    def main_calculate_step_left(p11, p12, p21, p22, p3, p13, p23, noncappingsidewallthick, cappingsidewallthick, tcp_pose_top):
        struct1 = analyze_touchpoints_only(p11, p12, p21, p22, p3)
        list1 = analyze_vertical_touchpoints(p11, p12, p13, p21, p22, p23, p3)
        #struct2 = calculate_DOtA_points_right(struct1, list1, chamferover)
        #validity = check_validity_right(struct1, struct2)
        struct2 = calculate_DAaU_step_left(struct1, list1, cappingsidewallthick, noncappingsidewallthick, tcp_pose_top)
        validity = check_validity_only(struct2)
        return struct2
    end

    # analyze_touchpoints_only()
    # it takes 5 arguments as points
    # it returns a struct containing: (pointintersect, heading1, heading2, heading3, l1delxunit, l1delyunit, l2delxunit, l2delyunit)
    #   FIND HEADINGS
    #for each heading, find the angle of the line with respect to the pos x axis. then add/subtract 90 degrees because you want to be perpendicular to that
    # so, heading1 finds the angle (from the +x axis) to the position pointing perpendicularly into the box.
    # we need to be +90 degrees of all 3 headings. (but we can ignore heading 2)
    def step_right_demo(struct1):
        pointintersect = struct1[0]
        x = pointintersect[0]
        y = pointintersect[1]
        z = pointintersect[2]
        heading1 = struct1[1]
        heading1adj1 = heading1 + pi/2 #(90 deg) (parrallel to edge not perpendicular into
        heading1adj2 = heading1adj1 - pi/2 #(90 deg) (from y+ not x+)
        # heading1 == heading1adj2. ok
        m1 = get_rotation_matrix_from_description("z", 1, heading1)
        # at this point we would multiply matrices, but there is only one matrix
        rxryrz = convert_matrix_to_axang(m1)
        point_demo = p[x, y, z, rxryrz[0], rxryrz[1], rxryrz[2]]
        popup(point_demo)
        movej(point_demo, a=1.4, v=0.1)
        popup(point_demo)
        ret = struct(point_demo = point_demo)
        return ret
    end

    # for a left seam step corner, calculate the toolpath points for a L (under) then Up and Around weld. for left obstacle step.
    def calculate_LtUA_step_left(struct1, listleans, rightwallthick, leftwallthick, tcp_pose_top):
        # get the stuff from the struct
        pointintersect = struct1[0]
        heading1 = struct1[1]
        heading2 = struct1[2]
        heading3 = struct1[3]
        l1delxunit = struct1[4]
        l1delyunit = struct1[5]
        l2delxunit = struct1[6]
        l2delyunit = struct1[7]

        # FIND THE POINTS ON THE LINES OF THE FIRST TURN PATH
        # find locations 8 inches away from  intersect point
        # CONST
        welddistance1 = 3 # first path first leg
        welddistance2 = 3 # first path second leg
        welddistance3 = 8 # vertical weld distance

        # inches
        wd1 = welddistance1 * 25.4 / 1000
        wd2 = welddistance2 * 25.4 / 1000
        wd3 = tcp_pose_top[2] - pointintersect[2] # the z distance from the corner to the top of the weld
        leftwallthickmm = leftwallthick * 25.4 / 1000 # in this step corner right, this is distance from left edge
        rightwallthickmm =  rightwallthick * 25.4 / 1000 # in this step corner right, this is distance from right edge


        # weld distance is the distance that it will weld. this will make it start at the z height that the user specified
        #wd1 = tcp_pose_top[2] - pointintersect[2] - zup # this will need to change for step corner right

        # point bottom (point of intersection of the two chamfers on the bottom)
        xbottom = pointintersect[0] + l1delxunit * leftwallthickmm + l2delxunit * rightwallthickmm
        ybottom = pointintersect[1] + l1delyunit * leftwallthickmm + l2delyunit * rightwallthickmm
        z = pointintersect[2]

        # point 1
        x = xbottom + l1delxunit * wd1
        y = ybottom + l1delyunit * wd1

        # get rxryrz for facing along towards the intersection. heading1 +90 deg - 90 deg
        m1 = get_rotation_matrix_from_description("z", 1, heading1)
        # at this point we would multiply matrices, but there is only one matrix
        rxryrz = convert_matrix_to_axang(m1)
        rx = rxryrz[0]
        ry = rxryrz[1]
        rz = rxryrz[2]
        point1 = p[x, y, z, rx, ry, rz]

        # point 2
        point2 = p[xbottom, ybottom, z, rx, ry, rz]

        # point 4
        # get rxryrz for facing along the second edge pointed toward the left. heading 3 + 90 - 90
        m1 = get_rotation_matrix_from_description("z", 1, heading3)
        # at this point we would multiply matrices, but there is only one matrix
        rxryrz = convert_matrix_to_axang(m1)
        rx = rxryrz[0]
        ry = rxryrz[1]
        rz = rxryrz[2]
        point4 = p[xbottom, ybottom, z, rx, ry, rz]

        # point 5
        x = xbottom + l2delxunit * wd2
        y = ybottom + l2delyunit * wd2
        point5 = p[x, y, z, rx, ry, rz]

        # now calculate the points of the Up Around
        # don't use heading3 at all.
        #point201 is at the chamfer intersection
        p201x = xbottom
        p201y = ybottom
        p201z = z

        # rxryrz is the same
        m1 = get_rotation_matrix_from_description("z", 1, heading1)
        # at this point we would multiply matrices, but there is only one matrix
        rxryrz = convert_matrix_to_axang(m1)
        rx = rxryrz[0]
        ry = rxryrz[1]
        rz = rxryrz[2]
        point201 = p[p201x, p201y, p201z, rx, ry, rz]

        # find side point (point on the side. where point 203 would be if roundoverdistance was 0)
        sidex = pointintersect[0] + l2delxunit * rightwallthickmm
        sidey = pointintersect[1] + l2delyunit * rightwallthickmm
        sidez = z

        # p202
        roundoverdistance = 0.05
        rod = roundoverdistance * 25.4 / 1000
        p202x = sidex + rod * l1delxunit
        p202y = sidey + rod * l1delyunit
        p202z = sidez
        point202 = p[p202x, p202y, p202z, rx, ry, rz]

        # p204 end of circle move
        p204x = sidex
        p204y = sidey
        p204z = sidez + rod

        # calculate rxryrz
        # first rotation: 90 degrees about x axis. positive direction. preheat is now facing up, and gun tip is pointed towards y- direction
        m1 = get_rotation_matrix_from_description("x", 1, 90 * pi / 180)
        # second rotation: rotate about z until you are facing into the front face. but only use heading 1
        # heading 1 is about 225 degrees. i need to go about 225 degrees. starting from y- instead of x+ cancels out the extra 90 degrees needed to go into face1 instead of parallel to face1
        m2 = get_rotation_matrix_from_description("z", 1, heading1)
        m3 = multiply_matrix(m2, m1)
        rxryrz = convert_matrix_to_axang(m3)
        rx = rxryrz[0]
        ry = rxryrz[1]
        rz = rxryrz[2]
        point204 = p[p204x, p204y, p204z, rx, ry, rz]

        #p205 (end of straight after cirlce move, before listleans
        straightlength = 1.0 # the moveP blend radius for the circle move was set to 1.0 mm in FloorCorner. we should be more than 2.0mm away from point2
        sld = straightlength * 25.4 / 1000
        point205 = p[p204x, p204y, sidez + sld, rx, ry, rz]

        #p206 (top of weld)
        p206x = sidex + wd3 * listleans[0]
        p206y = sidey + wd3 * listleans[1]
        p206z = sidez + wd3
        point206 = p[p206x, p206y, p206z, rx, ry, rz]

        # p203 (middle of turn)
        # we know that the angle is exactly 90 degrees
        delta = calc_rod_midpoint_90deg(rod)
        p203z = sidez + delta
        p203x = sidex + delta * l1delxunit
        p203y = sidey + delta * l1delyunit

        # calculate rxryrz
        m1 = get_rotation_matrix_from_description("x", 1, 45 * pi / 180)
        m2 = get_rotation_matrix_from_description("z", 1, heading1)
        m3 = multiply_matrix(m2, m1)
        rxryrz = convert_matrix_to_axang(m3)
        rx = rxryrz[0]
        ry = rxryrz[1]
        rz = rxryrz[2]
        point203 = p[p203x, p203y, p203z, rx, ry, rz]

        # form struct
        struct2 = struct(point1=point1, point2=point2, point4=point4, point5=point5, point201=point201, point202=point202, point203=point203, point204=point204, point205=point205, point206=point206)
        return struct2
    end

    # for a right step corner, calculate the toolpath points for a L (under) then Up and Around weld.
    def calculate_LtUA_step_right(struct1, list1, rightwallthick, leftwallthick, tcp_pose_top):
        # get the stuff from the struct
        pointintersect = struct1[0]
        heading1 = struct1[1]
        heading2 = struct1[2]
        heading3 = struct1[3]
        l1delxunit = struct1[4]
        l1delyunit = struct1[5]
        l2delxunit = struct1[6]
        l2delyunit = struct1[7]

        # FIND THE POINTS ON THE LINES OF THE FIRST TURN PATH
        # find locations 8 inches away from  intersect point
        # CONST
        welddistance1 = 3 # first path first leg
        welddistance2 = 3 # first path second leg
        welddistance3 = 8 # vertical weld distance

        # inches
        wd1 = welddistance1 * 25.4 / 1000
        wd2 = welddistance2 * 25.4 / 1000
        wd3 = welddistance3 * 25.4 / 1000
        leftwallthickmm = leftwallthick * 25.4 / 1000 # in this step corner right, this is distance from left edge
        rightwallthickmm =  rightwallthick * 25.4 / 1000 # in this step corner right, this is distance from right edge


        # weld distance is the distance that it will weld. this will make it start at the z height that the user specified
        #wd1 = tcp_pose_top[2] - pointintersect[2] - zup # this will need to change for step corner right

        # point bottom (point of intersection of the two chamfers on the bottom)
        xbottom = pointintersect[0] + l1delxunit * leftwallthickmm + l2delxunit * rightwallthickmm
        ybottom = pointintersect[1] + l1delyunit * leftwallthickmm + l2delyunit * rightwallthickmm
        z = pointintersect[2]

        # point 1
        x = xbottom + l1delxunit * wd1
        y = ybottom + l1delyunit * wd1

        m1 = get_rotation_matrix_from_description("z", 1, heading1)
        # at this point we would multiply matrices, but there is only one matrix
        rxryrz = convert_matrix_to_axang(m1)
        rx = rxryrz[0]
        ry = rxryrz[1]
        rz = rxryrz[2]
        point1 = p[x, y, z, rx, ry, rz]

        # point 2
        point2 = p[xbottom, ybottom, z, rx, ry, rz]

        # point 4
        m1 = get_rotation_matrix_from_description("z", 1, heading3)
        # at this point we would multiply matrices, but there is only one matrix
        rxryrz = convert_matrix_to_axang(m1)
        rx = rxryrz[0]
        ry = rxryrz[1]
        rz = rxryrz[2]
        point4 = p[xbottom, ybottom, z, rx, ry, rz]

        # point 5
        x = xbottom + l2delxunit * wd2
        y = ybottom + l2delyunit * wd2
        point5 = p[x, y, z, rx, ry, rz]


        # form struct
        struct2 = struct(point1=point1, point2=point2, point4=point4, point5=point5, point_1=point1, point_2=point1, point_3=point1, point_4=point1, point_5=point1)
        return struct2
    end

    # step corner with two seams on bottom face
    # vertical seam on left side of corner
    # Down Around and Under weld path, then Back Away
    # the first path uses backofhole TCP, the second path uses pretend_welder TCP
    def calculate_DAaU_step_left(struct1, listleans, rightwallthick, leftwallthick, tcp_pose_top):
        # get the stuff from the struct
        pointintersect = struct1[0]
        heading1 = struct1[1]
        heading2 = struct1[2]
        heading3 = struct1[3]
        l1delxunit = struct1[4]
        l1delyunit = struct1[5]
        l2delxunit = struct1[6]
        l2delyunit = struct1[7]

        # FIND THE POINTS ON THE LINES OF THE FIRST TURN PATH
        # find locations 8 inches away from  intersect point
        # CONST
        welddistance1 = 8 # first path first leg (down)
        welddistance2 = 3 # first path second leg (under) # inches
        welddistance3 = 3 # second path (back away) # inches

        wd1 = tcp_pose_top[2] - pointintersect[2] # the touchpoint minus the corner
        wd2 = welddistance2 * 25.4 / 1000
        wd3 = welddistance3 * 25.4 / 1000
        leftwallthickmm = leftwallthick * 25.4 / 1000 # in this step corner right, this is distance from left edge
        rightwallthickmm =  rightwallthick * 25.4 / 1000 # in this step corner right, this is distance from right edge

        # first, calculate the location of the bottom of the vertical chamfer (where point2 would be if there weren't any circle motion
        x = pointintersect[0] + l2delxunit * rightwallthickmm
        y = pointintersect[1] + l2delyunit * rightwallthickmm
        z = pointintersect[2]
        pointbottomvcham = p[x, y, z, 0, 0, 0]

        # calculate the rxryrz for facing the vertical chamfer, with the preheat down
        rxryrz = convert_heading_to_axang_preheatdown(heading3)
        rx = rxryrz[0]
        ry = rxryrz[1]
        rz = rxryrz[2]

        # next, calculate point1 using the listleans
        point1 = p[x + wd1*listleans[0], y + wd1*listleans[1], z + wd1, rx, ry, rz] # add in the listleans factor to follow the face of the box as we move up

        # calculate rxryrz for point2 and point2a (based on heading1). should be very similar to the heading for point1
        # only use the right side taps for circle move related things
        heading3basedh1 = heading1 - pi/2 # heading1 based on heading3
        rxryrz = convert_heading_to_axang_preheatdown(heading3basedh1)
        rx = rxryrz[0]
        ry = rxryrz[1]
        rz = rxryrz[2]

        # the round over distance is the distance from pointbottomvcham to point2 (which will be the same as distance to p4)
        roundoverdistance = 0.05
        rod = roundoverdistance * 25.4 / 1000
        point2 = p[x, y, z + rod, rx, ry, rz]

        # calculate point2a, which is directly above pointbottomvcham (used to straighten weldpath before circlemove)
        straightlength = 1.0 # the moveP blend radius for the circle move was set to 1.0 mm in FloorCorner. we should be more than 2.0mm away from point2
        sld = straightlength * 25.4 / 1000
        point2a = p[x, y, z + sld, rx, ry, rz]

        # calculate the rxryrz for facing the underneath section, with the preheat facing parallel to the right edge (rx and ry should be 0 because gun is facing up)
        # to convert heading1 into the description, subtract 90 degrees to go parallel  instead of into. subtract 90 degrees to start from y+ instead of x+
        heading1descr = heading1 - pi
        m1 = get_rotation_matrix_from_description("z", 1, heading1descr)
        rxryrz = convert_matrix_to_axang(m1)
        rx = rxryrz[0]
        ry = rxryrz[1]
        rz = rxryrz[2]

        # calculate point4
        p4x = x + l1delxunit * rod
        p4y = y + l1delyunit * rod
        point4 = p[p4x, p4y, z, rx, ry, rz]

        # calculate point5
        p5x = x + l1delxunit * wd2
        p5y = y + l1delyunit * wd2
        point5 = p[p5x, p5y, z, rx, ry, rz]

        # calculate point3
        # we know that the angle is exactly 90 degrees
        delta = calc_rod_midpoint_90deg(rod)
        p3z = z + delta
        p3x = x + delta * l1delxunit
        p3y = y + delta * l1delyunit

        # calculate rxryrz
        m1 = get_rotation_matrix_from_description("x", -1, 45 * pi / 180) # rotation 1: 45 degrees forward about x axis
        m2 = get_rotation_matrix_from_description("z", 1, heading1descr) # rotation 2
        m3 = multiply_matrix(m2, m1) #we rotate m1 first then m2, so we multiply in backwards order: 2 then 1
        rxryrz = convert_matrix_to_axang(m3)
        rx = rxryrz[0]
        ry = rxryrz[1]
        rz = rxryrz[2]
        point3 = p[p3x, p3y, p3z, rx, ry, rz]

        #todo: calculate trail out point

        # calculate back-away (points 201 and 202)
        pushtipforward = 0.006 # 6 millimeters forward. the tip needs to clear the capping wall's angled chamfer to not BONK when getting into position
        p201x = x + l1delxunit * leftwallthickmm + l2delxunit * pushtipforward
        p201y = y + l1delyunit * leftwallthickmm + l2delyunit * pushtipforward

        # calculate rxryrz
        m1 = get_rotation_matrix_from_description("z", 1, heading3)
        # minus pi/2 for the different start point. minus pi/2 for parallel not perpendicular into
        rxryrz = convert_matrix_to_axang(m1)
        rx = rxryrz[0]
        ry = rxryrz[1]
        rz = rxryrz[2]
        point201 = p[p201x, p201y, z, rx, ry, rz]

        # calculate point 202
        p202x = p201x + wd3 * l2delxunit
        p202y = p201y + wd3 * l2delyunit
        point202 = p[p202x, p202y, z, rx, ry, rz]

        struct2 = struct(point1=point1, point2a=point2a, point2=point2, point3=point3, point4=point4, point5=point5, point201=point201, point202=point202)
        return struct2
    end

    # step corner with two seams on bottom face
    # vertical seam on right side of corner
    # Down Around and Under weld path, then Back Away
    # the first path uses backofhole TCP, the second path uses pretend_welder TCP
    def calculate_DAaU_step_right(struct1, listleans, rightwallthick, leftwallthick, tcp_pose_top):
        # get the stuff from the struct
        pointintersect = struct1[0]
        heading1 = struct1[1]
        heading2 = struct1[2]
        heading3 = struct1[3]
        l1delxunit = struct1[4]
        l1delyunit = struct1[5]
        l2delxunit = struct1[6]
        l2delyunit = struct1[7]

        # FIND THE POINTS ON THE LINES OF THE FIRST TURN PATH
        # find locations 8 inches away from  intersect point
        # CONST
        welddistance1 = 8 # first path first leg (down)
        welddistance2 = 3 # first path second leg (under) # inches
        welddistance3 = 3 # second path (back away) # inches

        wd1 = tcp_pose_top[2] - pointintersect[2] # the touchpoint minus the corner
        wd2 = welddistance2 * 25.4 / 1000
        wd3 = welddistance3 * 25.4 / 1000
        leftwallthickmm = leftwallthick * 25.4 / 1000 # in this step corner right, this is distance from left edge
        rightwallthickmm =  rightwallthick * 25.4 / 1000 # in this step corner right, this is distance from right edge

        # first, calculate the location of the bottom of the vertical chamfer (where point2 would be if there weren't any circle motion
        x = pointintersect[0] + l1delxunit * leftwallthickmm
        y = pointintersect[1] + l1delyunit * leftwallthickmm
        z = pointintersect[2]
        pointbottomvcham = p[x, y, z, 0, 0, 0]

        # calculate the rxryrz for facing the vertical chamfer, with the preheat down
        rxryrz = convert_heading_to_axang_preheatdown(heading1)
        rx = rxryrz[0]
        ry = rxryrz[1]
        rz = rxryrz[2]

        # next, calculate point1 using the listleans
        point1 = p[x + wd1*listleans[0], y + wd1*listleans[1], z + wd1, rx, ry, rz] # add in the listleans factor to follow the face of the box as we move up

        # calculate rxryrz for point2 and point2a (based on heading3). should be very similar to the heading for point1
        # only use the left side taps for circle move related things
        heading1basedh3 = heading3 + pi/2 # heading1 based on heading3
        rxryrz = convert_heading_to_axang_preheatdown(heading1basedh3)
        rx = rxryrz[0]
        ry = rxryrz[1]
        rz = rxryrz[2]

        # the round over distance is the distance from pointbottomvcham to point2 (which will be the same as distance to p4)
        roundoverdistance = 0.05
        rod = roundoverdistance * 25.4 / 1000
        point2 = p[x, y, z + rod, rx, ry, rz]

        # calculate point2a, which is directly above pointbottomvcham (used to straighten weldpath before circlemove)
        straightlength = 1.0 # the moveP blend radius for the circle move was set to 1.0 mm in FloorCorner. we should be more than 2.0mm away from point2
        sld = straightlength * 25.4 / 1000
        point2a = p[x, y, z + sld, rx, ry, rz]


        # calculate the rxryrz for facing the underneath section, with the preheat facing parallel to the left edge (rx and ry should be 0 because gun is facing up)
        m1 = get_rotation_matrix_from_description("z", 1, heading3)
        rxryrz = convert_matrix_to_axang(m1)
        rx = rxryrz[0]
        ry = rxryrz[1]
        rz = rxryrz[2]

        # calculate point4
        p4x = x + l2delxunit * rod
        p4y = y + l2delyunit * rod
        point4 = p[p4x, p4y, z, rx, ry, rz]

        # calculate point5
        p5x = x + l2delxunit * wd2
        p5y = y + l2delyunit * wd2
        point5 = p[p5x, p5y, z, rx, ry, rz]

        # calculate point3
        # we know that the angle is exactly 90 degrees
        delta = calc_rod_midpoint_90deg(rod)
        p3z = z + delta
        p3x = x + delta * l2delxunit
        p3y = y + delta * l2delyunit

        # calculate rxryrz
        m1 = get_rotation_matrix_from_description("x", -1, 45 * pi / 180) # rotation 1: 45 degrees forward about x axis
        m2 = get_rotation_matrix_from_description("z", 1, heading3) # rotation 2
        m3 = multiply_matrix(m2, m1) #we rotate m1 first then m2, so we multiply in backwards order: 2 then 1
        rxryrz = convert_matrix_to_axang(m3)
        rx = rxryrz[0]
        ry = rxryrz[1]
        rz = rxryrz[2]
        point3 = p[p3x, p3y, p3z, rx, ry, rz]

        #todo: calculate trail out point

        # calculate back-away (points 201 and 202)
        pushtipforward = 0.006 # 6 millimeters forward. the tip needs to clear the capping wall's angled chamfer to not BONK when getting into position
        p201x = x + l2delxunit * rightwallthickmm + l1delxunit * pushtipforward
        p201y = y + l2delyunit * rightwallthickmm + l1delyunit * pushtipforward

        # calculate rxryrz
        m1 = get_rotation_matrix_from_description("z", 1, heading1 - pi)
        # minus pi/2 for the different start point. minus pi/2 for parallel not perpendicular into
        rxryrz = convert_matrix_to_axang(m1)
        rx = rxryrz[0]
        ry = rxryrz[1]
        rz = rxryrz[2]
        point201 = p[p201x, p201y, z, rx, ry, rz]

        # calculate point 202
        p202x = p201x + wd3 * l1delxunit
        p202y = p201y + wd3 * l1delyunit
        point202 = p[p202x, p202y, z, rx, ry, rz]

        struct2 = struct(point1=point1, point2a=point2a, point2=point2, point3=point3, point4=point4, point5=point5, point201=point201, point202=point202)
        return struct2
    end

    # given a round over distance (in mm), calculate (based on 90 degrees) the distance from corner (line intersection) to midpoint of arc
    # returns a value (in mm) that you need to move from line intersection to midpoint (actual distance will be this times sqrt(2))
    def calc_rod_midpoint_90deg(rod):
        # the factor is (1- 1/sqrt(2))
        factor = 0.292893
        ret = rod * factor
        return ret
    end

    # this is the main entry point for calculations, for Cover Corner.
    # it takes in the 4 touchpoints, analyzes the shape of the box.
    # returns the pathpoints
    # specifically for Around and Down then Straight (AtS)
    # specifically for left-sided boxes (vertical weld on left side of edge)
    # leftchoice is a boolean and deepcovercham is a boolean but leftwallthick, rightwallthick are decimals in inches.
    def main_calculate_cover(p11, p12, p21, p3, leftwallthick, rightwallthick, leftchoice, deepcovercham):
        struct1 = analyze_touchpoints_only_cover(p11, p12, p21, p3)
        if leftchoice:
            struct2 = calculate_AtS_points_cover_left(struct1, leftwallthick, rightwallthick, deepcovercham)
        else:
            struct2 = calculate_AtS_points_cover_right(struct1, leftwallthick, rightwallthick, deepcovercham)
        end
        #struct2 = calculate_DOtA_points_left_extended(struct1, list1, chamferover, chamferup, tcp_pose_top)
        #struct3 = check_validity_left(struct1, struct2)
        return struct2
    end

    def calculate_AtS_points_cover_left(struct1, leftwallthick, rightwallthick, deepcovercham):
        # get the stuff from the struct
        pointintersect = struct1[0]
        heading1 = struct1[1]
        heading2 = struct1[2]
        heading3 = struct1[3]
        l1delxunit = struct1[4]
        l1delyunit = struct1[5]
        l2delxunit = struct1[6]
        l2delyunit = struct1[7]

        # FIND THE POINTS ON THE LINES OF THE FIRST TURN PATH
        # find locations 8 inches away from  intersect point
        # CONST
        welddistance1 = 6 # first path first leg (down)
        welddistance2 = 3 # first path second leg (under) # inches
        welddistance3 = 6 # second path (back away) # inches

        wd1 = welddistance1 * 25.4 / 1000
        wd2 = welddistance2 * 25.4 / 1000
        wd3 = welddistance3 * 25.4 / 1000
        leftwallthickmm = leftwallthick * 25.4 / 1000 # in this step corner right, this is distance from left edge
        rightwallthickmm =  rightwallthick * 25.4 / 1000 # in this step corner right, this is distance from right edge
        if deepcovercham:
            deepchambumpmm = 0.09 * 25.4/1000 # if there is a deep chamfer on the cover, bump the welder inwards 0.09 more inches.
        else:
            deepchambumpmm = 0.0
        end

        # first, check if we need a lift column raise
        # (we do, because for maximum reach we want to make the lift pedestal be even with the top of the covers)
        zpi = pointintersect[2]
        if zpi > 0:
            liftcolumnzneeded = zpi * 1000.0 # the robot uses coordinates in meters, but the lift column uses coordinates in mm
            z = 0
        else:
            z = zpi
        end

        # first, calculate the location of the top of the vertical chamfer (where point2 would be if there weren't any circle motion)
        x = pointintersect[0] + l2delxunit * rightwallthickmm
        y = pointintersect[1] + l2delyunit * rightwallthickmm
        #z = pointintersect[2] # replaced by z of lift column (directly above)
        pointtopvcham = p[x, y, z, 0, 0, 0]

        # calculate the rxryrz for the gun when it's at point1
        # start with rxryrz = 0,0,0 (gun facing up, preheat facing y+ axis.
        # rotate it 180 degrees about x axis. gun facing down, preheat facing y- axis
        # rotate it about 45 degrees ccw about z axis. x+ to heading1 is about 135 degrees. so our angle is heading1 - 90 degrees
        m1 = get_rotation_matrix_from_description("x", -1, 180 * pi / 180) # rotation 1: 180 degrees forward about x axis
        m2 = get_rotation_matrix_from_description("z", 1, heading1 - pi/2) # rotation 2
        m3 = multiply_matrix(m2, m1) #we rotate m1 first then m2, so we multiply in backwards order: 2 then 1
        rxryrz = convert_matrix_to_axang(m3)
        rx = rxryrz[0]
        ry = rxryrz[1]
        rz = rxryrz[2]

        # next, calculate point1 (start point on top of cover welding towards corner)
        p1x = x + l1delxunit * wd1 + deepchambumpmm * l2delxunit
        p1y = y + l1delyunit * wd1 + deepchambumpmm * l2delyunit
        point1 = p[p1x, p1y, z, rx, ry, rz]

        # the round over distance is the distance from pointbottomvcham to point2 (which will be the same as distance to p4)
        roundoverdistance = 0.05
        rod = roundoverdistance * 25.4 / 1000
        p2x = x + l1delxunit * rod
        p2y = y + l1delyunit * rod
        point2 = p[p2x, p2y, z, rx, ry, rz]

        # make point2a, colinear between p1 and p2, which will be the place the welder shuts off during motion
        shutofftime = 1.5 # seconds. this is how soon to shut off extrusion before we hit point 2.
        if deepcovercham:
            speed = 6 # mm/s
            wtod = shutofftime * speed / 1000 #weldturnoffdistance
        else:
            speed = 10 # mm/s
            wtod = shutofftime * speed / 1000
        end
        p2ax = x + l1delxunit * wtod
        p2ay = y + l1delyunit * wtod
        point2a = p[p2ax, p2ay, z, rx, ry, rz]

        # calculate the rxryrz for facing the down the left side of the box
        # rotate about x 90 (forward). then rotate about z ~ 45 (ccw)
        m1 = get_rotation_matrix_from_description("x", -1, 90 * pi / 180)
        m2 = get_rotation_matrix_from_description("z", 1, heading1 - pi/2)
        m3 = multiply_matrix(m2, m1) #we rotate m1 first then m2, so we multiply in backwards order: 2 then 1
        rxryrz = convert_matrix_to_axang(m3)
        rx = rxryrz[0]
        ry = rxryrz[1]
        rz = rxryrz[2]

        # calculate point4
        point4 = p[x, y, z - rod, rx, ry, rz]

        # calculate point5
        point5 = p[x, y, z - wd2, rx, ry, rz]

        # calculate point3
        # we know that the angle is exactly 90 degrees
        delta = calc_rod_midpoint_90deg(rod)
        p3z = z - delta
        p3x = x + delta * l1delxunit
        p3y = y + delta * l1delyunit

        # calculate rxryrz
        m1 = get_rotation_matrix_from_description("x", -1, 135 * pi / 180) # rotation 1: 135 degrees forward about x axis
        m2 = get_rotation_matrix_from_description("z", 1, heading1 - pi/2)
        m3 = multiply_matrix(m2, m1) #we rotate m1 first then m2, so we multiply in backwards order: 2 then 1
        rxryrz = convert_matrix_to_axang(m3)
        rx3 = rxryrz[0]
        ry3 = rxryrz[1]
        rz3 = rxryrz[2]
        point3 = p[p3x, p3y, p3z, rx3, ry3, rz3]

        #todo: calculate trail out points
        botvcham = wd2 # where is the bottom of the v chamfer (z distance from top corner)
        tcpdiff = 14 # mm. the difference between backofhole tcp and welder tcp (tip)
        # calculate point5a (point101) (start of tilt back) (start of unflatten)
        dist = 1.5 * 25.4/1000 + tcpdiff/1000 # distance from botvcham
        p101x = x
        p101y = y
        p101z = z - wd2 + dist
        point101 = p[p101x, p101y, p101z, rx, ry, rz]

        # calculate point5b (point 102) (end of unflatten)
        dist = 0.5 * 25.4 / 1000
        tiltraise = 0.006
        p102x = x + l1delxunit * tiltraise * -1
        p102y = y + l1delyunit * tiltraise * -1
        p102z = z - wd2 + dist

        # calculate rxryrz
        tiltangledeg = 10 # ten degree angle of tilt
        m1 = get_rotation_matrix_from_description("x", -1, (90 + tiltangledeg) * pi / 180) # rotation 1: 135 degrees forward about x axis
        m2 = get_rotation_matrix_from_description("z", 1, heading1 - pi/2)
        m3 = multiply_matrix(m2, m1) #we rotate m1 first then m2, so we multiply in backwards order: 2 then 1
        rxryrz = convert_matrix_to_axang(m3)
        rx = rxryrz[0]
        ry = rxryrz[1]
        rz = rxryrz[2]
        point102 = p[p102x, p102y, p102z, rx, ry, rz]

        # calculate point 5c (point 103) (end of smear)
        dist = -2 * 25.4/1000
        point103 = p[p102x, p102y, z - wd2 + dist, rx, ry, rz]

        # calculate back-away (points 201 and 202)
        pushtipforward = 0.006 # 6 millimeters forward. the tip needs to clear the capping wall's angled chamfer to not BONK when getting into position
        p201x = x + l1delxunit * (leftwallthickmm + deepchambumpmm) + l2delxunit * pushtipforward
        p201y = y + l1delyunit * (leftwallthickmm + deepchambumpmm) + l2delyunit * pushtipforward

        # calculate rxryrz
        # rotate 180 degrees about x. then rotate (90 deg + heading3 degrees) about z ccw
        m1 = get_rotation_matrix_from_description("x", -1, 180 * pi / 180)
        m2 = get_rotation_matrix_from_description("z", 1, heading3 + pi/2)
        m3 = multiply_matrix(m2, m1) #we rotate m1 first then m2, so we multiply in backwards order: 2 then 1
        rxryrz = convert_matrix_to_axang(m3)
        rx = rxryrz[0]
        ry = rxryrz[1]
        rz = rxryrz[2]
        point201 = p[p201x, p201y, z, rx, ry, rz]

        # calculate point 201's preheat
        pushtipforward2 = 0.012 - pushtipforward + deepchambumpmm # 12 mm forward to clear the existing extrudant (but still have the extrudant from this extrusion join the existing). subtract from previous to make it constant even if you change pushtipforward1
        preheatdistance = 0.010 # 10 mm . above what it would be pushed down
        point201a = p[p201x, p201y, z + preheatdistance, rx, ry, rz]
        p201bx = p201x + l2delxunit * pushtipforward2
        p201by = p201y + l2delyunit * pushtipforward2
        point201b = p[p201bx, p201by, z + preheatdistance, rx, ry, rz]
        point201c = p[p201bx, p201by, z, rx, ry, rz]

        # calculate point 202
        p202x = p201x + wd3 * l2delxunit
        p202y = p201y + wd3 * l2delyunit
        point202 = p[p202x, p202y, z, rx, ry, rz]

        struct2 = struct(point1=point1, point2=point2, point3=point3, point4=point4, point5=point5, point201=point201, point202=point202, point201a=point201a, point201b=point201b, point201c=point201c, point2a=point2a, point101=point101, point102=point102, point103=point103)
        return struct2
    end

    def calculate_AtS_points_cover_right(struct1, leftwallthick, rightwallthick, deepcovercham):
        # get the stuff from the struct
        pointintersect = struct1[0]
        heading1 = struct1[1]
        heading2 = struct1[2]
        heading3 = struct1[3]
        l1delxunit = struct1[4]
        l1delyunit = struct1[5]
        l2delxunit = struct1[6]
        l2delyunit = struct1[7]

        # FIND THE POINTS ON THE LINES OF THE FIRST TURN PATH
        # find locations 8 inches away from  intersect point
        # CONST
        welddistance1 = 6 # first path first leg (down)
        welddistance2 = 3 # first path second leg (under) # inches
        welddistance3 = 6 # second path (back away) # inches

        wd1 = welddistance1 * 25.4 / 1000
        wd2 = welddistance2 * 25.4 / 1000
        wd3 = welddistance3 * 25.4 / 1000
        leftwallthickmm = leftwallthick * 25.4 / 1000 # in this step corner right, this is distance from left edge
        rightwallthickmm =  rightwallthick * 25.4 / 1000 # in this step corner right, this is distance from right edge

        if deepcovercham:
            deepchambumpmm = 0.09 * 25.4/1000 # if there is a deep chamfer on the cover, bump the welder inwards 0.09 more inches.
        else:
            deepchambumpmm = 0.0
        end

        # first, check if we need a lift column raise
        # (we do, because for maximum reach we want to make the lift pedestal be even with the top of the covers)
        zpi = pointintersect[2]
        if zpi > 0:
            liftcolumnzneeded = zpi * 1000.0 # the robot uses coordinates in meters, but the lift column uses coordinates in mm
            z = 0
        else:
            z = zpi
        end

        # first, calculate the location of the top of the vertical chamfer (where point2 would be if there weren't any circle motion)
        x = pointintersect[0] + l1delxunit * leftwallthickmm
        y = pointintersect[1] + l1delyunit * leftwallthickmm
        #z = pointintersect[2] # replaced by z of lift column (directly above)
        pointtopvcham = p[x, y, z, 0, 0, 0]

        # calculate the rxryrz for the gun when it's at point1
        # start with rxryrz = 0,0,0 (gun facing up, preheat facing y+ axis.
        # rotate it 180 degrees about x axis. gun facing down, preheat facing y- axis
        # rotate it about 135 degrees ccw about z axis. x+ to heading3 is about 225 degrees. so our angle is heading3 - 90 degrees
        m1 = get_rotation_matrix_from_description("x", -1, 180 * pi / 180) # rotation 1: 180 degrees forward about x axis
        m2 = get_rotation_matrix_from_description("z", 1, heading3 - pi/2) # rotation 2
        m3 = multiply_matrix(m2, m1) #we rotate m1 first then m2, so we multiply in backwards order: 2 then 1
        rxryrz = convert_matrix_to_axang(m3)
        rx = rxryrz[0]
        ry = rxryrz[1]
        rz = rxryrz[2]

        # next, calculate point1 (start point on top of cover welding towards corner)
        p1x = x + l2delxunit * wd1 + deepchambumpmm * l1delxunit
        p1y = y + l2delyunit * wd1 + deepchambumpmm * l1delyunit
        point1 = p[p1x, p1y, z, rx, ry, rz]

        # the round over distance is the distance from pointbottomvcham to point2 (which will be the same as distance to p4)
        roundoverdistance = 0.05
        rod = roundoverdistance * 25.4 / 1000
        p2x = x + l2delxunit * rod
        p2y = y + l2delyunit * rod
        point2 = p[p2x, p2y, z, rx, ry, rz]

        # make point2a, colinear between p1 and p2, which will be the place the welder shuts off during motion
        shutofftime = 1.5 # seconds. this is how soon to shut off extrusion before we hit point 2.
        if deepcovercham:
            speed = 6 # mm/s
            wtod = shutofftime * speed / 1000 #weldturnoffdistance
        else:
            speed = 10 # mm/s
            wtod = shutofftime * speed / 1000
        end
        p2ax = x + l2delxunit * wtod
        p2ay = y + l2delyunit * wtod
        point2a = p[p2ax, p2ay, z, rx, ry, rz]

        # calculate the rxryrz for facing the down the right side of the box
        # rotate about x 90 (forward). then rotate about z ~ 135 (ccw)
        m1 = get_rotation_matrix_from_description("x", -1, 90 * pi / 180)
        m2 = get_rotation_matrix_from_description("z", 1, heading3 - pi/2)
        m3 = multiply_matrix(m2, m1) #we rotate m1 first then m2, so we multiply in backwards order: 2 then 1
        rxryrz = convert_matrix_to_axang(m3)
        rx = rxryrz[0]
        ry = rxryrz[1]
        rz = rxryrz[2]

        # calculate point4
        point4 = p[x, y, z - rod, rx, ry, rz]

        # calculate point5
        point5 = p[x, y, z - wd2, rx, ry, rz]

        # calculate point3
        # we know that the angle is exactly 90 degrees
        delta = calc_rod_midpoint_90deg(rod)
        p3z = z - delta
        p3x = x + delta * l2delxunit
        p3y = y + delta * l2delyunit

        # calculate rxryrz
        m1 = get_rotation_matrix_from_description("x", -1, 135 * pi / 180) # rotation 1: 135 degrees forward about x axis
        m2 = get_rotation_matrix_from_description("z", 1, heading3 - pi/2)
        m3 = multiply_matrix(m2, m1) #we rotate m1 first then m2, so we multiply in backwards order: 2 then 1
        rxryrz = convert_matrix_to_axang(m3)
        rx3 = rxryrz[0]
        ry3 = rxryrz[1]
        rz3 = rxryrz[2]
        point3 = p[p3x, p3y, p3z, rx3, ry3, rz3]

        #todo: calculate trail out point
        botvcham = wd2 # where is the bottom of the v chamfer (z distance from top corner)
        tcpdiff = 14 # mm. the difference between backofhole tcp and welder tcp (tip)
        # calculate point5a (point101) (start of tilt back) (start of unflatten)
        dist = 1.5 * 25.4/1000 + tcpdiff/1000 # distance from botvcham
        p101x = x
        p101y = y
        p101z = z - wd2 + dist
        point101 = p[p101x, p101y, p101z, rx, ry, rz]

        # calculate point5b (point 102) (end of unflatten)
        dist = 0.5 * 25.4 / 1000
        tiltraise = 0.006
        p102x = x + l2delxunit * tiltraise * -1
        p102y = y + l2delyunit * tiltraise * -1
        p102z = z - wd2 + dist

        # calculate rxryrz
        tiltangledeg = 10 # ten degree angle of tilt
        m1 = get_rotation_matrix_from_description("x", -1, (90 + tiltangledeg) * pi / 180) # rotation 1: 135 degrees forward about x axis
        m2 = get_rotation_matrix_from_description("z", 1, heading3 - pi/2)
        m3 = multiply_matrix(m2, m1) #we rotate m1 first then m2, so we multiply in backwards order: 2 then 1
        rxryrz = convert_matrix_to_axang(m3)
        rx = rxryrz[0]
        ry = rxryrz[1]
        rz = rxryrz[2]
        point102 = p[p102x, p102y, p102z, rx, ry, rz]

        # calculate point 5c (point 103) (end of smear)
        dist = -2 * 25.4/1000
        point103 = p[p102x, p102y, z - wd2 + dist, rx, ry, rz]

        # calculate back-away (points 201 and 202)
        pushtipforward = 0.006 # 6 millimeters forward. the tip needs to clear the capping wall's angled chamfer to not BONK when getting into position
        p201x = x + l2delxunit * (rightwallthickmm + deepchambumpmm) + l1delxunit * pushtipforward
        p201y = y + l2delyunit * (rightwallthickmm + deepchambumpmm) + l1delyunit * pushtipforward

        # calculate rxryrz
        # rotate 180 degrees about x. then rotate (90 deg + heading1 degrees) about z ccw
        m1 = get_rotation_matrix_from_description("x", -1, 180 * pi / 180)
        m2 = get_rotation_matrix_from_description("z", 1, heading1 + pi/2)
        m3 = multiply_matrix(m2, m1) #we rotate m1 first then m2, so we multiply in backwards order: 2 then 1
        rxryrz = convert_matrix_to_axang(m3)
        rx = rxryrz[0]
        ry = rxryrz[1]
        rz = rxryrz[2]
        point201 = p[p201x, p201y, z, rx, ry, rz]

        # calculate point 201's preheat
        pushtipforward2 = 0.012 - pushtipforward + deepchambumpmm # 12 mm forward to clear the existing extrudant (but still have the extrudant from this extrusion join the existing). subtract from previous to make it constant even if you change pushtipforward1
        preheatdistance = 0.010 # 10 mm . above what it would be pushed down
        point201a = p[p201x, p201y, z + preheatdistance, rx, ry, rz]
        p201bx = p201x + l1delxunit * pushtipforward2
        p201by = p201y + l1delyunit * pushtipforward2
        point201b = p[p201bx, p201by, z + preheatdistance, rx, ry, rz]
        point201c = p[p201bx, p201by, z, rx, ry, rz]

        # calculate point 202
        p202x = p201x + wd3 * l1delxunit
        p202y = p201y + wd3 * l1delyunit
        point202 = p[p202x, p202y, z, rx, ry, rz]

        struct2 = struct(point1=point1, point2=point2, point3=point3, point4=point4, point5=point5, point201=point201, point202=point202, point201a=point201a, point201b=point201b, point201c=point201c, point2a=point2a, point101=point101, point102=point102, point103=point103)
        return struct2
    end

    def main_calculate_cover_straight(p11, p12, p21, p22, sidewallthick, leftpoint, rightpoint, deepcovercham):
        struct1 = analyze_touchpoints_only_cover_straight(p11, p12, p21, p22, leftpoint)
        struct2 = calculate_straight_points_cover(struct1, sidewallthick, leftpoint, rightpoint, deepcovercham)
        #struct2 = calculate_DOtA_points_left_extended(struct1, list1, chamferover, chamferup, tcp_pose_top)
        #struct3 = check_validity_left(struct1, struct2)
        return struct2

    end

    # calculates the line of intersection of the sidewall plane (assumed vertical) and the cover plane (assumed perpendicular to sidewall plane)
    # returns a struct containing point0 (point on the intersection line, same y as leftpoint) and 3 components of the unit vector left to right and 2 components of the other direction in 2d
    def analyze_touchpoints_only_cover_straight(p11, p12, p21, p22, leftpoint):
        # calculate slope of sidewall in x-y plane
        # get the raw points from the first line
        l1p1x=p11[0]
        l1p1y=p11[1]
        l1p2x=p12[0]
        l1p2y=p12[1]

        # equate the first line in 2d space
        ml1 = (l1p2y-l1p1y) / (l1p2x-l1p1x)

        # b = y - mx
        bl1 = l1p1y - ml1 * l1p1x

        # calculate the cover plane
        # if two planes are perpendicular, then their normal vectors must be perpendicular.
        # the first planes normal vector is n1, which is taken from the equation of the plane ax + by + cz = d -> <a, b, c>
        # the second plane's normal vector is perpendicular to all vectors contained in the plane
        # p21 to p22 is a vector v contained within plane 2.
        # n2 is normal to both n1 AND v. to achieve a vector that is normal to both, take the cross product

        # plane 1 (y = mx + b) -> (b = -mx +1y +0z)
        n1 = [-1 * ml1, 1, 0]

        # v=P2−P1=(x2−x1,y2−y1,z2−z1)
        v = [p21[0]-p22[0], p21[1]-p22[1], p21[2]-p22[2]]

        #v n2 = cross product of n1 and v
        n2x = n1[1]*v[2] - n1[2]*v[1]
        n2y = n1[2]*v[0] - n1[0]*v[2]
        n2z = n1[0]*v[1] - n1[1]*v[0]
        n2 = [n2x, n2y, n2z]

        # find the d of the second plane
        # n2x * x + n2y * y + n2z * z = d0
        d = n2x * p21[0] + n2y * p21[1] + n2z * p21[2]

        # find the intersection line of the two planes
        # find the direction vector of that line by taking the cross product of the normal vector of those two planes
        v3x = n1[1]*n2[2] - n1[2]*n2[1]
        v3y = n1[2]*n2[0] - n1[0]*n2[2]
        v3z = n1[0]*n2[1] - n1[1]*n2[0]
        v3 = [v3x, v3y, v3z]

        # normalize the vector so the magnitude is 1
        magnitude2 = v3x * v3x + v3y * v3y + v3z * v3z
        magnitude = sqrt(magnitude2)
        v3xunit = v3x/magnitude
        v3yunit = v3y/magnitude
        v3zunit = v3z/magnitude

        # make sure it is going the right way (from left to right). make sure the v3yunit is positive
        if v3yunit < 0:
            v3xunit = v3xunit * -1
            v3yunit = v3yunit * -1
            v3zunit = v3zunit * -1
        end

        # next we have to find a point on the line by setting one of the dimensions and solving the system of equations
        # i will pick the y value of the left teach point
        y = leftpoint[1]
        # plane 1: -ml1 * x + 1 * y + 0 * z = bl1
        # -ml1 * x = bl1 - y
        x = (bl1 - y)/ (-1 * ml1)
        # plane 2: d = n2x * x + n2y * y + n2z * z
        # (d - n2x * x - n2y * y) = n2z * z
        z = (d - n2x * x - n2y * y) / n2z

        # make point0 into a pose
        point0 = p[x, y, z, 0, 0, 0]

        # find heading of main line
        heading1 = convert_uv_to_heading(v3xunit, v3yunit)

        # make a unit vector perpendicular to this one in the xy plane pointing x -. will be used to move over the chamfer distance
        ml2 = -1 / ml1
        # y = ml2 * x + unknownB
        # vector = [1, ml2]
        mag2 = 1 + ml2 * ml2
        mag = sqrt(mag2)
        v4xunit = 1 / mag
        v4yunit = ml2 / mag
        # switch is to the x direction is negative
        v4xunit = -1 * v4xunit
        v4yunit = -1 * v4yunit

        ret = struct(point0=point0, v3xunit=v3xunit, v3yunit=v3yunit, v3zunit=v3zunit, heading1=heading1, v4xunit=v4xunit, v4yunit=v4yunit)
        return ret
    end

    def calculate_straight_points_cover(struct1, sidewallthick, leftpointteach, rightpointteach, deepcovercham):
        # get the stuff
        point0 = struct1[0]
        p0x = point0[0]
        p0y = point0[1]
        p0z = point0[2]
        v3xunit = struct1[1]
        v3yunit = struct1[2]
        v3zunit = struct1[3]
        heading1 = struct1[4]
        v4xunit = struct1[5]
        v4yunit = struct1[6]
        sidewallthick = sidewallthick
        lpy = leftpointteach[1]
        rpy = rightpointteach[1]

        # first, check if we need a lift column raise
        # (we do, because for maximum reach we want to make the lift pedestal be even with the top of the covers)
        zpi = p0z
        if zpi > 0:
            liftcolumnzneeded = zpi * 1000.0 # the robot uses coordinates in meters, but the lift column uses coordinates in mm
            coverz = 0
        else:
            coverz = zpi
        end

        if deepcovercham:
            deepchambumpmm = 0.09 * 25.4/1000 # if there is a deep chamfer on the cover, bump the welder inwards 0.09 more inches.
        else:
            deepchambumpmm = 0.0
        end

        # calculate pointtopvcham
        chamferover = sidewallthick * 25.4 / 1000.0 + deepchambumpmm
        tiltraise = 0.006 # 6 mm raise needed for the tip to clear the plane during tiltback
        x = p0x + v4xunit * chamferover
        y = p0y + v4yunit * chamferover
        z = coverz + tiltraise

        # calculate rxryrz for tilted back
        # 3 rotations to make this happen.
        # start point is straight up with the preheat pointed in the +y direction.
        # first rotation is 180 degrees about x direction. gun is now pointing straight down with preheat facing -y direction
        m1 = get_rotation_matrix_from_description("x", 1, 180 * pi / 180)
        # second rotation is a 10 degree turn about the x axis (negative direction)
        m2 = get_rotation_matrix_from_description("x", -1, 10 * pi / 180)
        # third rotation is about 180 degrees about the z axis. starting from the -y axis, go until you get to heading1. that will equal heading1 plus 90 degrees
        m3 = get_rotation_matrix_from_description("z", 1, pi/2 + heading1)
        # combine them by multiplying m3 * m2 * m1
        # matrix multiplication is not commutative but it IS associative, so you can do this whichever order
        m4 = multiply_matrix(m2, m1)
        m5 = multiply_matrix(m3, m4)
        rxryrzt = convert_matrix_to_axang(m5)
        rxt = rxryrzt[0]
        ryt = rxryrzt[1]
        rzt = rxryrzt[2]
        pointtopvcham = p[x, y, z, rxt, ryt, rzt]

        # calculate point1 (preheat)
        dist = -1 * 25.4 / 1000.0 # move back 1 inch from
        p1x = x + dist * v3xunit
        p1y = y + dist * v3yunit
        p1z = z + dist * v3zunit
        point1 = p[p1x, p1y, p1z, rxt, ryt, rzt]

        # calculate point2 (start of flatten)
        dist = 0.5 * 25.4 / 1000.0  # half an inch past the top of v chamfer
        p2x = x + dist * v3xunit
        p2y = y + dist * v3yunit
        p2z = z + dist * v3zunit
        point2 = p[p2x, p2y, p2z, rxt, ryt, rzt]

        # calculate rxryrz for nontilted
        # first rotation is 180 degrees about x direction. gun is now pointing straight down with preheat facing -y direction
        m1 = get_rotation_matrix_from_description("x", 1, 180 * pi / 180)
        # third rotation is about 180 degrees about the z axis. starting from the -y axis, go until you get to heading1. that will equal heading1 plus 90 degrees
        m3 = get_rotation_matrix_from_description("z", 1, pi/2 + heading1)
        m5 = multiply_matrix(m3, m1)
        rxryrz = convert_matrix_to_axang(m5)
        rx = rxryrz[0]
        ry = rxryrz[1]
        rz = rxryrz[2]

        # calculate point3 (end of flatten)
        dist = 1.5 * 25.4 / 1000.0  # 1.5 inches past top of v chamfer
        p3x = x + dist * v3xunit
        p3y = y + dist * v3yunit
        p3z = coverz + dist * v3zunit
        point3 = p[p3x, p3y, p3z, rx, ry, rz]

        # calculate distance between leftpoint and rightpoint
        # we have the y distance. we need to find the total distance.
        # the unit vector (v3) should have a magnitude of 1. that's what analyze_touchpoints_only_cover_straight() calculated.
        # so the total distance is y distance * 1 / v3yunit
        ydist = rpy - lpy
        totdist = ydist / v3yunit

        # calculate pointtopvcham2
        x2 = x + v3xunit * totdist
        y2 = y + v3yunit * totdist
        z2 = z + v3zunit * totdist

        # calculate point4 (start of unflatten)
        dist = -1.5 * 25.4 / 1000.0
        p4x = x2 + v3xunit * dist
        p4y = y2 + v3yunit * dist
        p4z = z2 + v3zunit * dist - tiltraise
        point4 = p[p4x, p4y, p4z, rx, ry, rz]

        # calculate point5 (end of unflatten)
        dist = -0.5 * 25.4 / 1000.0
        p5x = x2 + v3xunit * dist
        p5y = y2 + v3yunit * dist
        p5z = z2 + v3zunit * dist
        point5 = p[p5x, p5y, p5z, rxt, ryt, rzt]

        # calculate point6 (end of smear)
        dist = 2 * 25.4 / 1000.0
        p6x = x2 + v3xunit * dist
        p6y = y2 + v3yunit * dist
        p6z = z2 + v3zunit * dist
        point6 = p[p6x, p6y, p6z, rxt, ryt, rzt]


        # return struct
        ret = struct(pointtopvcham=pointtopvcham, point1=point1, point2=point2, point3=point3, point4=point4, point5=point5, point6=point6)
        return ret


    end

    def main_calculate_floor_straight(p11, p12, p21, p22, floorthick, leftpoint, rightpoint):
        struct1 = analyze_touchpoints_only_cover_straight(p11, p12, p21, p22, leftpoint)
        struct2 = calculate_straight_points_floor(struct1, floorthick, leftpoint, rightpoint)
        #struct2 = calculate_DOtA_points_left_extended(struct1, list1, chamferover, chamferup, tcp_pose_top)
        #struct3 = check_validity_left(struct1, struct2)
        return struct2

    end

    # the path for welding a floor straight weld with v chisels on both sides.
    # start at the right side and move left.
    def calculate_straight_points_floor(struct1, floorthick, leftpointteach, rightpointteach):
        # get the stuff
        point0 = struct1[0]
        p0x = point0[0]
        p0y = point0[1]
        p0z = point0[2]
        v3xunit = struct1[1]
        v3yunit = struct1[2]
        v3zunit = struct1[3]
        heading1 = struct1[4]
        v4xunit = struct1[5]
        v4yunit = struct1[6]
        lpy = leftpointteach[1]
        rpy = rightpointteach[1]

        # first, check if we need a lift column raise
        # (we do not, because the floors are low)
        zpi = p0z
        floorz = zpi

        # calculate pointtopvcham (left point) (tilted and tiltraised)
        chamferup = floorthick * 25.4 / 1000.0
        tiltraise = 0.006 # 6 mm raise needed for the tip to clear the plane during tiltback
        # on this one, move the tiltraise distance sideways (towards robot) and the chamferover distance up
        x = p0x + v4xunit * tiltraise * -1
        y = p0y + v4yunit * tiltraise * -1
        z = floorz + chamferup

        # calculate rxryrz for tilted back
        # 3 rotations to make this happen.
        # start point is straight up with the preheat pointed in the +y direction.
        # first rotation is 90 degrees about y axis. positive direction. gun is now pointing in the x+ direction with preheat facing +y direction
        m1 = get_rotation_matrix_from_description("y", 1, 90 * pi / 180)
        # second rotation is about 180 degrees about the z axis. heading1 plus 90 degrees. gun is now pointing directly into the sidewall
        m2 = get_rotation_matrix_from_description("z", 1, pi/2 + heading1)
        # third rotation is 10 degrees about the z axis. gun is now tilted back 10 degrees from the sidewall
        m3 = get_rotation_matrix_from_description("z", 1, 10 * pi / 180)
        # combine them by multiplying m3 * m2 * m1
        # matrix multiplication is not commutative but it IS associative, so you can do this whichever order
        m4 = multiply_matrix(m2, m1)
        m5 = multiply_matrix(m3, m4)
        rxryrzt = convert_matrix_to_axang(m5)
        rxt = rxryrzt[0]
        ryt = rxryrzt[1]
        rzt = rxryrzt[2]
        # the non tilted angle is just m4
        rxryrz = convert_matrix_to_axang(m4)
        rx = rxryrz[0]
        ry = rxryrz[1]
        rz = rxryrz[2]
        pointtopvcham = p[x, y, z, rxt, ryt, rzt]

        # calculate distance between leftpoint and rightpoint
        # we have the y distance. we need to find the total distance.
        # the unit vector (v3) should have a magnitude of 1. that's what analyze_touchpoints_only_cover_straight() calculated.
        # so the total distance is y distance * 1 / v3yunit
        ydist = rpy - lpy
        totdist = ydist / v3yunit

        # calculate pointtopvcham2 (right point) (tilted and tiltraised)
        x2 = x + v3xunit * totdist
        y2 = y + v3yunit * totdist
        z2 = z + v3zunit * totdist
        pointtopvcham2 = p[x2, y2, z2, rxt, ryt, rzt]

        # calculate point1 (preheat)
        dist = 1 * 25.4 / 1000.0 # move back 1 inch from ptvc2 (in this case back means positive)
        p1x = x2 + dist * v3xunit
        p1y = y2 + dist * v3yunit
        p1z = z2 + dist * v3zunit
        point1 = p[p1x, p1y, p1z, rxt, ryt, rzt]

        # calculate point2 (start of flatten)
        dist = -0.5 * 25.4 / 1000.0  # half an inch past the top of v chamfer
        p2x = x2 + dist * v3xunit
        p2y = y2 + dist * v3yunit
        p2z = z2 + dist * v3zunit
        point2 = p[p2x, p2y, p2z, rxt, ryt, rzt]

        # calculate point3 (end of flatten)
        dist = -1.5 * 25.4 / 1000.0  # 1.5 inches past top of v chamfer
        p3x = x2 + dist * v3xunit + tiltraise * v4xunit
        p3y = y2 + dist * v3yunit + tiltraise * v4yunit
        p3z = z2 + dist * v3zunit
        point3 = p[p3x, p3y, p3z, rx, ry, rz]

        # calculate point4 (start of unflatten)
        dist = 1.5 * 25.4 / 1000.0
        p4x = x + v3xunit * dist + tiltraise * v4xunit
        p4y = y + v3yunit * dist + tiltraise * v4yunit
        p4z = z + v3zunit * dist
        point4 = p[p4x, p4y, p4z, rx, ry, rz]

        # calculate point5 (end of unflatten)
        dist = 0.5 * 25.4 / 1000.0
        p5x = x + v3xunit * dist
        p5y = y + v3yunit * dist
        p5z = z + v3zunit * dist
        point5 = p[p5x, p5y, p5z, rxt, ryt, rzt]

        # calculate point6 (end of smear)
        dist = -2 * 25.4 / 1000.0
        p6x = x + v3xunit * dist
        p6y = y + v3yunit * dist
        p6z = z + v3zunit * dist
        point6 = p[p6x, p6y, p6z, rxt, ryt, rzt]

        # return struct
        ret = struct(pointtopvcham=pointtopvcham, point1=point1, point2=point2, point3=point3, point4=point4, point5=point5, point6=point6)
        return ret

    end

    # this function determines the starting touchpoints for homing in on cover lt geometry
    # includes two points above the cover lt, closer to the robot than the lt, facing down
    def get_coverlt_homing_pathpoints(leftpoint, rightpoint):
        # get the teach position points
        lpx = leftpoint[0]
        lpy = leftpoint[1]
        lpz = leftpoint[2]
        rpx = rightpoint[0]
        rpy = rightpoint[1]
        rpz = rightpoint[2]

        # specify the distances from (in meters)
        d0 = 0.05 # how far from the cover to approach from
        d1 = 0.03 # how far the touchpints are pushed closer to the robot
        d2 = 0.00 # how far inwards the touchpoints are pushed

        # rxryrz
        rxryrz = [0.334, 3.124, 0]
        rx = rxryrz[0]
        ry = rxryrz[1]
        rz = rxryrz[2]

        # calculate the points
        ph1 = p[lpx + d1, lpy + d2, lpz + d0, rx, ry, rz] # left side approach
        ph2 = p[rpx + d1, rpy - d2, rpz + d0, rx, ry, rz] # right side approach

        ret = struct(ph1=ph1, ph2=ph2)
        is_robot_at_reachable_spot(leftpoint, ret)
        return ret
    end

    def main_calculate_cover_lt(p11, p12, leftpoint, rightpoint):
        struct1 = analyze_touchpoints_only_cover_lt(p11, p12, leftpoint, rightpoint)
        struct2 = calculate_points_cover_lt(struct1)
        #struct2 = calculate_DOtA_points_left_extended(struct1, list1, chamferover, chamferup, tcp_pose_top)
        #struct3 = check_validity_left(struct1, struct2)
        return struct2

    end

    def analyze_touchpoints_only_cover_lt(p11, p12, leftpoint, rightpoint):
        # calculate the slope of the groove in xy plane
        l1p1x = leftpoint[0]
        l1p1y = leftpoint[1]
        l1p2x = rightpoint[0]
        l1p2y = rightpoint[1]

        # equate the first line in 2d space
        ml1 = (l1p2y-l1p1y) / (l1p2x-l1p1x)

        # b = y - mx
        bl1 = l1p1y - ml1 * l1p1x

        # zraise (how much the z value changes from left point to right point
        zraise = p12[2] - p11[2]

        #get the calcpoints
        leftcalcpoint = [leftpoint[0], leftpoint[1], p11[2]]
        rightcalcpoint = [rightpoint[0], rightpoint[1], p12[2]]
        # get the vector from a to b
        vec = [rightcalcpoint[0] - leftcalcpoint[0], rightcalcpoint[1] - leftcalcpoint[1], rightcalcpoint[2] - leftcalcpoint[2]]
        # get the unit vector in 3d
        mag3d = sqrt(vec[0]*vec[0]+vec[1]*vec[1]+vec[2]*vec[2])
        vec3dunit = [vec[0]/mag3d, vec[1]/mag3d, vec[2]/mag3d]
        # get the unit vector in 2d
        mag2d = sqrt(vec[0]*vec[0]+vec[1]*vec[1])
        vec2dunit = [vec[0]/mag2d, vec[1]/mag2d]
        # get the heading
        heading1 = convert_uv_to_heading(vec2dunit[0], vec2dunit[1])

        ret = struct(leftcalcpoint=leftcalcpoint, rightcalcpoint=rightcalcpoint, vxunit=vec3dunit[0], vyunit=vec3dunit[1], vzunit=vec3dunit[2], heading1=heading1)
        return ret
    end

    def calculate_points_cover_lt(struct1):
        # get the stuff from struct
        leftcalcpoint = struct1[0]
        x = leftcalcpoint[0]
        y = leftcalcpoint[1]
        z = leftcalcpoint[2]
        rightcalcpoint = struct1[1]
        x2 = rightcalcpoint[0]
        y2 = rightcalcpoint[1]
        z2 = rightcalcpoint[2]
        v3xunit = struct1[2]
        v3yunit = struct1[3]
        v3zunit = struct1[4]
        heading1 = struct1[5]

        # first calculate rxryrz f normal and tiltback
        # calculate rxryrz for tilted back
        # 3 rotations to make this happen.
        # start point is straight up with the preheat pointed in the +y direction.
        # first rotation is 180 degrees about x direction. gun is now pointing straight down with preheat facing -y direction
        m1 = get_rotation_matrix_from_description("x", 1, 180 * pi / 180)
        # second rotation is a 10 degree turn about the x axis (negative direction)
        m2 = get_rotation_matrix_from_description("x", -1, 10 * pi / 180)
        # third rotation is about 180 degrees about the z axis. starting from the -y axis, go until you get to heading1. that will equal heading1 plus 90 degrees
        m3 = get_rotation_matrix_from_description("z", 1, pi/2 + heading1)
        # combine them by multiplying m3 * m2 * m1
        # matrix multiplication is not commutative but it IS associative, so you can do this whichever order
        m4 = multiply_matrix(m2, m1)
        m5 = multiply_matrix(m3, m4)
        rxryrzt = convert_matrix_to_axang(m5)
        rxt = rxryrzt[0]
        ryt = rxryrzt[1]
        rzt = rxryrzt[2]

        # calculate rxryrz for nontilted
        # first rotation is 180 degrees about x direction. gun is now pointing straight down with preheat facing -y direction
        m1 = get_rotation_matrix_from_description("x", 1, 180 * pi / 180)
        # third rotation is about 180 degrees about the z axis. starting from the -y axis, go until you get to heading1. that will equal heading1 plus 90 degrees
        m3 = get_rotation_matrix_from_description("z", 1, pi/2 + heading1)
        m5 = multiply_matrix(m3, m1)
        rxryrz = convert_matrix_to_axang(m5)
        rx = rxryrz[0]
        ry = rxryrz[1]
        rz = rxryrz[2]

        tiltraise = 0.006 # 6 mm raise needed for the tip to clear the plane during tiltback

        # calculate points 1-3
        # calculate point1 (preheat)
        dist = -1 * 25.4 / 1000.0 # move back 1 inch from
        p1x = x + dist * v3xunit
        p1y = y + dist * v3yunit
        p1z = z + dist * v3zunit + tiltraise
        point1 = p[p1x, p1y, p1z, rxt, ryt, rzt]

        # calculate point2 (start of flatten)
        dist = 0.5 * 25.4 / 1000.0  # half an inch past the top of v chamfer
        p2x = x + dist * v3xunit
        p2y = y + dist * v3yunit
        p2z = z + dist * v3zunit + tiltraise
        point2 = p[p2x, p2y, p2z, rxt, ryt, rzt]

        # calculate point3 (end of flatten)
        dist = 1.5 * 25.4 / 1000.0  # 1.5 inches past top of v chamfer
        p3x = x + dist * v3xunit
        p3y = y + dist * v3yunit
        p3z = z + dist * v3zunit
        point3 = p[p3x, p3y, p3z, rx, ry, rz]

        # calculate points 4-6
        # calculate point4 (start of unflatten)
        dist = -1.5 * 25.4 / 1000.0
        p4x = x2 + v3xunit * dist
        p4y = y2 + v3yunit * dist
        p4z = z2 + v3zunit * dist
        point4 = p[p4x, p4y, p4z, rx, ry, rz]

        # calculate point5 (end of unflatten)
        dist = -0.5 * 25.4 / 1000.0
        p5x = x2 + v3xunit * dist
        p5y = y2 + v3yunit * dist
        p5z = z2 + v3zunit * dist + tiltraise
        point5 = p[p5x, p5y, p5z, rxt, ryt, rzt]

        # calculate point6 (end of smear)
        dist = 2 * 25.4 / 1000.0
        p6x = x2 + v3xunit * dist
        p6y = y2 + v3yunit * dist
        p6z = z2 + v3zunit * dist + tiltraise
        point6 = p[p6x, p6y, p6z, rxt, ryt, rzt]

        # return struct
        ret = struct(pointtopvcham=leftcalcpoint, point1=point1, point2=point2, point3=point3, point4=point4, point5=point5, point6=point6)
        return ret

    end
    $ 329 "path_pre≔get_coverlt_homing_pathpoints(tcp_pose_left,tcp_pose_right)"
    global path_pre=get_coverlt_homing_pathpoints(tcp_pose_left,tcp_pose_right)
    $ 330 "ph1≔path_pre[0]"
    global ph1=path_pre[0]
    $ 331 "ph2≔path_pre[1]"
    global ph2=path_pre[1]
    $ 334 "MoveL"
    $ 335 "Direction: Base Z+"
    global move_thread_flag_335=0
    thread move_thread_335():
      enter_critical
      move_thread_flag_335 = 1
      local towardsPos=calculate_point_to_move_towards(p[0.0,0.0,0.0,0.0,0.0,0.0], [0.0,0.0,1.0], 0.1)
      movel(towardsPos, a=1.2, v=0.25)
      move_thread_flag_335 = 2
      exit_critical
    end
    move_thread_flag_335 = 0
    move_thread_han_335 = run move_thread_335()
    while (True):
      sleep(1.0E-10)
      if (move_thread_flag_335 > 1):
        join move_thread_han_335
        $ 336 "Until (distance)"
        break
      end
      sync()
    end
    $ 337 "MoveL"
    $ 338 "ph2" "breakAfter"
    movel(ph2, a=0.2, v=0.25)
    $ 339 "MoveL"
    $ 340 "Direction: Base Z-"
    global move_thread_flag_340=0
    thread move_thread_340():
      enter_critical
      move_thread_flag_340 = 1
      local towardsPos=calculate_point_to_move_towards(p[0.0,0.0,0.0,0.0,0.0,0.0], [0.0,0.0,-1.0], 1000.0)
      movel(towardsPos, a=0.1, v=0.02)
      move_thread_flag_340 = 2
      exit_critical
    end
    move_thread_flag_340 = 0
    move_thread_han_340 = run move_thread_340()
    while (True):
      local targetTcpDirection=get_target_tcp_speed()
      local stepsToRetract=tool_contact(direction=targetTcpDirection)
      if (stepsToRetract > 0):
        kill move_thread_han_340
        stopl(3.0)
        local backTrackMovement=get_actual_joint_positions_history(stepsToRetract)
        local contactPose=get_forward_kin(backTrackMovement)
        local posDir=[targetTcpDirection[0],targetTcpDirection[1],targetTcpDirection[2]]
        local retractTo=contactPose
        if (norm(posDir) > 1e-6):
          local normalizedPosDir=normalize(posDir)
          local additionalRetraction=p[normalizedPosDir[0] * 0.0, normalizedPosDir[1] * 0.0, normalizedPosDir[2] * 0.0, 0, 0, 0]
          retractTo = pose_sub(contactPose, additionalRetraction)
        end
        movel(retractTo, a=3.0, v=0.1)
        $ 341 "Until (tool_contact_detection)"
        break
      end
      sync()
    end
    $ 342 "p12≔get_actual_tcp_pose()"
    global p12= get_actual_tcp_pose ()
    $ 343 "MoveL"
    $ 344 "ph2" "breakAfter"
    movel(ph2, a=1.2, v=0.25)
    $ 345 "ph1" "breakAfter"
    movel(ph1, a=1.2, v=0.25)
    $ 346 "MoveL"
    $ 347 "Direction: Base Z-"
    global move_thread_flag_347=0
    thread move_thread_347():
      enter_critical
      move_thread_flag_347 = 1
      local towardsPos=calculate_point_to_move_towards(p[0.0,0.0,0.0,0.0,0.0,0.0], [0.0,0.0,-1.0], 1000.0)
      movel(towardsPos, a=0.1, v=0.02)
      move_thread_flag_347 = 2
      exit_critical
    end
    move_thread_flag_347 = 0
    move_thread_han_347 = run move_thread_347()
    while (True):
      local targetTcpDirection=get_target_tcp_speed()
      local stepsToRetract=tool_contact(direction=targetTcpDirection)
      if (stepsToRetract > 0):
        kill move_thread_han_347
        stopl(3.0)
        local backTrackMovement=get_actual_joint_positions_history(stepsToRetract)
        local contactPose=get_forward_kin(backTrackMovement)
        local posDir=[targetTcpDirection[0],targetTcpDirection[1],targetTcpDirection[2]]
        local retractTo=contactPose
        if (norm(posDir) > 1e-6):
          local normalizedPosDir=normalize(posDir)
          local additionalRetraction=p[normalizedPosDir[0] * 0.0, normalizedPosDir[1] * 0.0, normalizedPosDir[2] * 0.0, 0, 0, 0]
          retractTo = pose_sub(contactPose, additionalRetraction)
        end
        movel(retractTo, a=3.0, v=0.1)
        $ 348 "Until (tool_contact_detection)"
        break
      end
      sync()
    end
    $ 356 "p11≔get_actual_tcp_pose()"
    global p11= get_actual_tcp_pose ()
    $ 357 "MoveJ"
    $ 358 "ph1" "breakAfter"
    movej(ph1, a=1.3962634015954636, v=1.0471975511965976)
    $ 359 "MoveJ"
    $ 360 "ph1" "breakAfter"
    movej(ph1, a=1.3962634015954636, v=1.0471975511965976)
    $ 361 "MoveJ"
    $ 362 "Waypoint_2" "breakAfter"
    movej(get_inverse_kin(Waypoint_2_p, qnear=Waypoint_2_q), a=1.3962634015954636, v=1.0471975511965976)
    $ 363 "Home"
    movej([-3.266929759358355, -1.2139462677784536, 1.5878387874396154, 1.1069165929565088, -0.0023738326664366483, -1.7891447305770605], a=1.3962634015954636, v=1.0471975511965976)
  end
  $ 2 "BeforeStart"
  $ 90 "'for this, dont have to worry about the normal stuff. just send it up and home'"
  # 'for this, dont have to worry about the normal stuff. just send it up and home'
  $ 91 "Cover Safe Home Folder"
  $ 92 "'if robot is not at home, send it back to home safely'"
  # 'if robot is not at home, send it back to home safely'
  $ 93 "'make sure the tcp is welder'"
  # 'make sure the tcp is welder'
  $ 94 "Set"
  set_tcp(p[-0.0095,-0.328,0.10573,1.2092,-1.2092,1.2092])
  $ 95 "sp≔get_actual_tcp_pose()"
  global sp= get_actual_tcp_pose ()
  $ 96 "MoveL"
  $ 97 "sp" "breakAfter"
  movel(sp, a=1.2, v=0.25)
  $ 98 "'if first move is to a variable, skip automove'"
  # 'if first move is to a variable, skip automove'
  $ 99 "'turn off welder'"
  # 'turn off welder'
  # begin: URCap Program Node
  #   Source: WireTank Serial, 4.9.0, WireTank, LLC
  #   Type: WireTank Serial
  $ 100 "Serial Bridge uR0"
  SerialResponse = WTSerialBridge.send_command("/dev/ttyUSB0",1200, 8, "None", "One", "None", 1000, "None", "None", [252,82,48], False)
  # end: URCap Program Node
  $ 101 "Set DO[0]=Off"
  set_standard_digital_out(0, False)
  $ 102 "jp≔get_actual_joint_positions()"
  global jp= get_actual_joint_positions ()
  $ 103 "If sp[0]>0.600"
  if (sp[0]>0.600):
    $ 104 "'if x > 600 then above then home'"
    # 'if x > 600 then above then home'
    $ 105 "MoveJ"
    $ 107 "Waypoint_76" "breakAfter"
    movej(get_inverse_kin(Waypoint_76_p, qnear=Waypoint_76_q), a=1.3962634015954636, v=1.0471975511965976)
    $ 108 "Home"
    movej([-3.266929759358355, -1.2139462677784536, 1.5878387874396154, 1.1069165929565088, -0.0023738326664366483, -1.7891447305770605], a=1.3962634015954636, v=1.0471975511965976)
  else:
    $ 109 "Else" "noBreak"
    $ 110 "Popup: retreating to home"
    popup("retreating to home", "Message", False, False, blocking=True)
    $ 111 "MoveL"
    $ 112 "Direction: Base Z+"
    global move_thread_flag_112=0
    thread move_thread_112():
      enter_critical
      move_thread_flag_112 = 1
      local towardsPos=calculate_point_to_move_towards(p[0.0,0.0,0.0,0.0,0.0,0.0], [0.0,0.0,1.0], 0.1)
      movel(towardsPos, a=1.2, v=0.25)
      move_thread_flag_112 = 2
      exit_critical
    end
    move_thread_flag_112 = 0
    move_thread_han_112 = run move_thread_112()
    while (True):
      sleep(1.0E-10)
      if (move_thread_flag_112 > 1):
        join move_thread_han_112
        $ 113 "Until (distance)"
        break
      end
      sync()
    end
    $ 117 "'insert logic for how to get back to oldhome'"
    # 'insert logic for how to get back to oldhome'
    $ 118 "'finish with oldhome then above then home'"
    # 'finish with oldhome then above then home'
    $ 123 "Home"
    movej([-3.266929759358355, -1.2139462677784536, 1.5878387874396154, 1.1069165929565088, -0.0023738326664366483, -1.7891447305770605], a=1.3962634015954636, v=1.0471975511965976)
  end
  $ 364 "Thread_1"
  thread Thread_1():
    $ 365 "Loop  True "
    while (  True  ):
      $ 366 "If freedrive_m_var≟ True "
      if (freedrive_m_var ==   True  ):
        $ 367 "freedrive_mode()"
        freedrive_mode()
        $ 368 "free_dr_already≔ True "
        global free_dr_already=  True
      else:
        $ 369 "Else" "noBreak"
        $ 370 "If free_dr_already"
        if (free_dr_already):
          $ 371 "end_freedrive_mode()"
          end_freedrive_mode()
        end
      end
      $ 372 "sync()"
      sync()
    end
  end
  threadId_Thread_1 = run Thread_1()
  $ 125 "Robot Program"
  $ 126 "'start of main program'"
  # 'start of main program'
  $ 127 "Set"
  set_tcp(p[-0.0095,-0.328,0.10573,1.2092,-1.2092,1.2092])
  $ 128 "Home"
  movej([-3.266929759358355, -1.2139462677784536, 1.5878387874396154, 1.1069165929565088, -0.0023738326664366483, -1.7891447305770605], a=1.3962634015954636, v=1.0471975511965976)
  $ 129 "Script: analyze_touchpoints.script"
  # this file creates the function for analyzing touchpoints
  # define pi
  pi = 3.1415926535
  # initialize a lift column extension needed of 0.0
  global liftcolumnzneeded = 0.0

  # this is the main entry point for calculations.
  # it takes in the 5 points, analyzes the shape of the box, and then calculates path points and returns them
  # specifically for Down, Over, then Around (DOtA)
  # specifically for right-sided boxes (vertical weld on right side of edge)
  def main_calculate_right(p11, p12, p21, p22, p3, p13, p23, chamferover):
      struct1 = analyze_touchpoints_only(p11, p12, p21, p22, p3)
      list1 = analyze_vertical_touchpoints(p11, p12, p13, p21, p22, p23, p3)
      struct2 = calculate_DOtA_points_right(struct1, list1, chamferover)
      validity = check_validity_right(struct1, struct2)
      return struct2
  end

  # this is the main entry point for calculations.
  # it takes in the 5 points, analyzes the shape of the box, and then calculates path points and returns them
  # specifically for Down, Over, then Around (DOtA)
  # specifically for left-sided boxes (vertical weld on left side of edge)
  def main_calculate_left(p11, p12, p21, p22, p3, p13, p23, chamferover):
      struct1 = analyze_touchpoints_only(p11, p12, p21, p22, p3)
      list1 = analyze_vertical_touchpoints(p11, p12, p13, p21, p22, p23, p3)
      struct2 = calculate_DOtA_points_left(struct1, list1, chamferover)
      validity = check_validity_left(struct1, struct2)
      return struct2
  end

  # this is the main entry point for calculations, for Floor Corner Extended.
  # it takes in the 7 touchpoints, analyzes the shape of the box.
  # takes in the user defined point for the top of the weld (tcp_pose_top) and then calculates path points
  # loopingly tries to calculate the extension along the sidewall that fulfills get_inverse_kin_has_solution() and provides the farthest extension possible
  # returns the pathpoints
  # specifically for Down, Over, then Around (DOtA)
  # specifically for right-sided boxes (vertical weld on right side of edge)
  def main_calculate_right_extended(p11, p12, p21, p22, p3, p13, p23, chamferover, chamferup, tcp_pose_top):
      struct1 = analyze_touchpoints_only(p11, p12, p21, p22, p3)
      list1 = analyze_vertical_touchpoints(p11, p12, p13, p21, p22, p23, p3)
      struct2 = calculate_DOtA_points_right_extended(struct1, list1, chamferover, chamferup, tcp_pose_top)
      struct3 = check_validity_right(struct1, struct2)
      return struct3
  end

  # this is the main entry point for calculations, for Floor Corner Extended.
  # it takes in the 7 touchpoints, analyzes the shape of the box.
  # takes in the user defined point for the top of the weld (tcp_pose_top) and then calculates path points
  # loopingly tries to calculate the extension along the sidewall that fulfills get_inverse_kin_has_solution() and provides the farthest extension possible
  # returns the pathpoints
  # specifically for Down, Over, then Around (DOtA)
  # specifically for left-sided boxes (vertical weld on left side of edge)
  def main_calculate_left_extended(p11, p12, p21, p22, p3, p13, p23, chamferover, chamferup, tcp_pose_top):
      struct1 = analyze_touchpoints_only(p11, p12, p21, p22, p3)
      list1 = analyze_vertical_touchpoints(p11, p12, p13, p21, p22, p23, p3)
      struct2 = calculate_DOtA_points_left_extended(struct1, list1, chamferover, chamferup, tcp_pose_top)
      struct3 = check_validity_left(struct1, struct2)
      return struct3
  end

  # it takes 5 arguments as points
  # it returns a struct containing: (pointintersect, pointapproach1, pointapproach2, point1, point2, point3, point4, point5, pointreturn1, heading1, heading2, heading3, path2r1, path2r2, path2l1, path2l2)
  # specifically for Around then Up (AtU)
  def analyze_touchpoints(p11, p12, p21, p22, p3):
    # FIND THE INTERSECTION
    # comment get the z
    zcoord=p3[2]

    # get the raw points from the first line
    l1p1x=p11[0]
    l1p1y=p11[1]
    l1p2x=p12[0]
    l1p2y=p12[1]

    # equate the first line in 2d space
    ml1 = (l1p2y-l1p1y) / (l1p2x-l1p1x)

    # b = y - mx
    bl1 = l1p1y - ml1 * l1p1x

    # get the raw points from the second line
    l2p1x=p21[0]
    l2p1y=p21[1]
    l2p2x=p22[0]
    l2p2y=p22[1]

    # equate the second line in 2d space
    ml2 = (l2p2y-l2p1y) / (l2p2x-l2p1x)

    # b = y - mx
    bl2 = l2p1y - ml2 * l2p1x


    # find the intersection of the two lines
    # m1x+b1 = m2x+b2
    # m1x - m2x = b2 - b1
    # x = (b2-b1) / (m1-m2)
    xintersect = (bl2-bl1) / (ml1-ml2)
    yintersect = ml1 * xintersect + bl1

    #FIND THE VECTORS
    #define a vector from the intersection to the second point on the first line
    l1delxfull = l1p2x - xintersect
    l1delyfull = l1p2y - yintersect

    l1delmag = sqrt(l1delxfull*l1delxfull + l1delyfull*l1delyfull)

    l1delxunit = l1delxfull / l1delmag
    l1delyunit = l1delyfull / l1delmag

    #define a vector from the intersection to the second point on the second line
    l2delxfull = l2p2x - xintersect
    l2delyfull = l2p2y - yintersect

    l2delmag = sqrt(l2delxfull*l2delxfull + l2delyfull*l2delyfull)

    l2delxunit = l2delxfull / l2delmag
    l2delyunit = l2delyfull / l2delmag

    # FIND THE FOUR POINTS ON THE LINES
    # find locations 8 inches away from  intersect point
    # CONST
    welddistance = 8
    roundoverdistance = 0.05
    zup = .375
    # inches
    wd = welddistance * 25.4 / 1000
    rod = roundoverdistance * 25.4 / 1000
    zup = zup * 25.4 / 1000

    # now we have the unit vector. extend the weld distance from the intersection
    x = xintersect + l1delxunit * wd
    y = yintersect + l1delyunit * wd
    z = zcoord + zup

    point1 = p[x,y,z,1.570796,0,0] # dummy orientation for now

    x = xintersect + l1delxunit * rod
    y = yintersect + l1delyunit * rod

    point2 = p[x,y,z,1.570796,0,0]

    # now we have the unit vector. extend the weld distance from the intersection
    x = xintersect + l2delxunit * wd
    y = yintersect + l2delyunit * wd

    point5 = p[x,y,z,0,-1.570796,0]

    x = xintersect + l2delxunit * rod
    y = yintersect + l2delyunit * rod

    point4 = p[x,y,z,0,-1.570796,0]

    #DEFINE APPROACH POINTS
    pointintersect = p[xintersect,yintersect,zcoord,0,0,0]
    pointapproach1 = p[xintersect+0.1,yintersect+0.1,z,1.570796,0,0]
    pointapproach2 = p[point1[0], point1[1]+0.1, point1[2], point1[3], point1[4], point1[5]]
    pointreturn1 = p[point5[0]+0.1, point5[1], point5[2], point5[3], point5[4], point5[5]]

    #FIND HEADINGS
    #for each heading, find the angle of the line with respect to the pos x axis. then add/subtract 90 degrees because you want to be perpendicular to that
    headingvector1 = convert_uv_to_heading(l1delxunit, l1delyunit)
    headingvector2 = convert_uv_to_heading(l2delxunit, l2delyunit)
    # find halfway heading
    heading2 = (headingvector1 + headingvector2)/2
    # find headings that the robot should face while traveling, perpendicular to the vectors of the sides of the box
    heading1 = headingvector1 + pi/2
    heading3 = headingvector2 - pi/2

    #FIND POINT 3
    #see if we have to / can find point 3
    findpoint3 = True
    if roundoverdistance == 0:
      findpoint3 = False
    end
    if findpoint3:
      # i need to find the point3 such that the arc from p2 to p3 to p4 is tangent to p1-p2 and p4-p5. making this a smooth path will be good
      # the direction of movement is from pointintersect in the direction of heading2
      # how much movement though? this will depend on whether it is actually a 90 degree angle or not.
      # first, find the perpendicular lines through points 2 and 4
      perp2 = find_perpendicular_line(ml1, point2[0], point2[1])
      perp4 = find_perpendicular_line(ml2, point4[0], point4[1])
      # next, find the intersection of those two lines
      perpintersect = find_intersection(perp2[0], perp2[1], perp4[0], perp4[1])
      radiusofcircle = distance_between(perpintersect[0], perpintersect[1], 0, point2[0], point2[1], 0)
      # find a vector the direction of heading2
      uvx = cos(heading2)
      uvy = sin(heading2)
      # compute point3. pass in negative radius because the direction is into the tank but we want to move from the intersection out to the rounded edge
      point3coords = add_vectordistance_to_point(perpintersect[0], perpintersect[1], z, uvx, uvy, 0, -1 * radiusofcircle)
      point3 = p[point3coords[0], point3coords[1], point3coords[2], 0, 0, 0]
    end

    #APPLY ACTUAL RXRYRZ TO POINTS
    # convert the headings to rxryrz and insert those values into the relevant points
    rxryrz = convert_heading_to_axang(heading1)
    rx = rxryrz[0]
    ry = rxryrz[1]
    rz = rxryrz[2]
    pointapproach1 = p[pointapproach1[0], pointapproach1[1], pointapproach1[2], rx, ry, rz]
    pointapproach2 = p[pointapproach2[0], pointapproach2[1], pointapproach2[2], rx, ry, rz]
    point1 = p[point1[0], point1[1], point1[2], rx, ry, rz]
    point2 = p[point2[0], point2[1], point2[2], rx, ry, rz]
    rxryrz = convert_heading_to_axang(heading2)
    rx = rxryrz[0]
    ry = rxryrz[1]
    rz = rxryrz[2]
    if findpoint3:
      point3 = p[point3[0], point3[1], point3[2], rx, ry, rz]
    else:
      point3 = point2
    end
    rxryrz = convert_heading_to_axang(heading3)
    rx = rxryrz[0]
    ry = rxryrz[1]
    rz = rxryrz[2]
    point4 = p[point4[0], point4[1], point4[2], rx, ry, rz]
    point5 = p[point5[0], point5[1], point5[2], rx, ry, rz]
    pointreturn1 = p[pointreturn1[0], pointreturn1[1], pointreturn1[2], rx, ry, rz]

    #find path2 (the part that goes up)
    four_vertical_points = find_vertical_points(pointintersect, l1delxunit, l1delyunit, l2delxunit, l2delyunit, zup, wd, heading1, heading3)
    path2r1 = four_vertical_points[0]
    path2r2 = four_vertical_points[1]
    path2l1 = four_vertical_points[2]
    path2l2 = four_vertical_points[3]

    #RETURN STRUCT
    ret = struct(pointintersect=pointintersect, pointapproach1=pointapproach1, pointapproach2=pointapproach2, point1=point1, point2=point2, point3=point3, point4=point4, point5=point5, pointreturn1=pointreturn1, heading1=heading1, heading2=heading2, heading3=heading3, path2r1=path2r1, path2r2=path2r2, path2l1=path2l1, path2l2=path2l2)
    return ret
  end

  # based on a Corner Homing 45 Cover pattern of touchpoints
  # this uses those touchpoints to create a representation of the corner in 3d robot space.
  def analyze_touchpoints_only_cover(p11, p12, p21, p3):
      zcoord=p3[2]

      # get the raw points from the first line
      l1p1x=p11[0]
      l1p1y=p11[1]
      l1p2x=p12[0]
      l1p2y=p12[1]

      # equate the first line in 2d space
      ml1 = (l1p2y-l1p1y) / (l1p2x-l1p1x)

      # b = y - mx
      bl1 = l1p1y - ml1 * l1p1x

      # get the raw points from the second line
      l2p1x=p21[0]
      l2p1y=p21[1]

      # equate the second line in 2d space
      # ml2 = opposite reciprocal of ml1 (because they are perpendicular) (assume perpendicular to make calculation of weldpath much easier)
      ml2 = -1 / ml1

      # b = y - mx
      bl2 = l2p1y - ml2 * l2p1x

      # find the intersection of the two lines
      # m1x+b1 = m2x+b2
      # m1x - m2x = b2 - b1
      # x = (b2-b1) / (m1-m2)
      xintersect = (bl2-bl1) / (ml1-ml2)
      yintersect = ml1 * xintersect + bl1

      pointintersect = p[xintersect,yintersect,zcoord,0,0,0]

      #FIND THE VECTORS
      #define a vector from the intersection to the second point on the first line
      l1delxfull = l1p2x - xintersect
      l1delyfull = l1p2y - yintersect

      l1delmag = sqrt(l1delxfull*l1delxfull + l1delyfull*l1delyfull)

      l1delxunit = l1delxfull / l1delmag
      l1delyunit = l1delyfull / l1delmag

      #define a vector from the intersection to the second point on the second line
      l2delxfull = l2p1x - xintersect
      l2delyfull = l2p1y - yintersect

      l2delmag = sqrt(l2delxfull*l2delxfull + l2delyfull*l2delyfull)

      l2delxunit = l2delxfull / l2delmag
      l2delyunit = l2delyfull / l2delmag

      #FIND HEADINGS
      #for each heading, find the angle of the line with respect to the pos x axis. this line is from pointintersect and along each edge of the corner
      heading1 = convert_uv_to_heading(l1delxunit, l1delyunit)
      heading3 = convert_uv_to_heading(l2delxunit, l2delyunit)
      # find halfway heading
      heading2 = (heading1 + heading3)/2

      #RETURN STRUCT
      ret = struct(pointintersect=pointintersect, heading1=heading1, heading2=heading2, heading3=heading3, l1delxunit=l1delxunit, l1delyunit=l1delyunit, l2delxunit=l2delxunit, l2delyunit=l2delyunit)
      return ret
  end

  # it takes 5 arguments as points
  # it returns a struct containing: (pointintersect, heading1, heading2, heading3, l1delxunit, l1delyunit, l2delxunit, l2delyunit)
  def analyze_touchpoints_only(p11, p12, p21, p22, p3):
    # FIND THE INTERSECTION
    # comment get the z
    zcoord=p3[2]

    # get the raw points from the first line
    l1p1x=p11[0]
    l1p1y=p11[1]
    l1p2x=p12[0]
    l1p2y=p12[1]

    # equate the first line in 2d space
    ml1 = (l1p2y-l1p1y) / (l1p2x-l1p1x)

    # b = y - mx
    bl1 = l1p1y - ml1 * l1p1x

    # get the raw points from the second line
    l2p1x=p21[0]
    l2p1y=p21[1]
    l2p2x=p22[0]
    l2p2y=p22[1]

    # equate the second line in 2d space
    ml2 = (l2p2y-l2p1y) / (l2p2x-l2p1x)

    # b = y - mx
    bl2 = l2p1y - ml2 * l2p1x


    # find the intersection of the two lines
    # m1x+b1 = m2x+b2
    # m1x - m2x = b2 - b1
    # x = (b2-b1) / (m1-m2)
    xintersect = (bl2-bl1) / (ml1-ml2)
    yintersect = ml1 * xintersect + bl1

    pointintersect = p[xintersect,yintersect,zcoord,0,0,0]

    #FIND THE VECTORS
    #define a vector from the intersection to the second point on the first line
    l1delxfull = l1p2x - xintersect
    l1delyfull = l1p2y - yintersect

    l1delmag = sqrt(l1delxfull*l1delxfull + l1delyfull*l1delyfull)

    l1delxunit = l1delxfull / l1delmag
    l1delyunit = l1delyfull / l1delmag

    #define a vector from the intersection to the second point on the second line
    l2delxfull = l2p2x - xintersect
    l2delyfull = l2p2y - yintersect

    l2delmag = sqrt(l2delxfull*l2delxfull + l2delyfull*l2delyfull)

    l2delxunit = l2delxfull / l2delmag
    l2delyunit = l2delyfull / l2delmag

    #FIND HEADINGS
    #for each heading, find the angle of the line with respect to the pos x axis. then add/subtract 90 degrees because you want to be perpendicular to that
    headingvector1 = convert_uv_to_heading(l1delxunit, l1delyunit)
    headingvector2 = convert_uv_to_heading(l2delxunit, l2delyunit)
    # find halfway heading
    heading2 = (headingvector1 + headingvector2)/2
    # find headings that the robot should face while traveling, perpendicular to the vectors of the sides of the box
    heading1 = headingvector1 + pi/2
    heading3 = headingvector2 - pi/2

    #RETURN STRUCT
    ret = struct(pointintersect=pointintersect, heading1=heading1, heading2=heading2, heading3=heading3, l1delxunit=l1delxunit, l1delyunit=l1delyunit, l2delxunit=l2delxunit, l2delyunit=l2delyunit)
    return ret
  end

  # given a struct from analyze_touchpoints_only(), calculate the points
  # for right, for non-extended
  def calculate_DOtA_points_right(struct1, listleans, chamferover):
      # get the stuff from the struct
      pointintersect = struct1[0]
      heading1 = struct1[1]
      heading2 = struct1[2]
      heading3 = struct1[3]
      l1delxunit = struct1[4]
      l1delyunit = struct1[5]
      l2delxunit = struct1[6]
      l2delyunit = struct1[7]

      # FIND THE POINTS ON THE LINES OF THE FIRST TURN PATH
      # find locations 8 inches away from  intersect point
      # CONST
      welddistance1 = 8 # vertical weld distance
      welddistance2 = 6 # first path second leg
      welddistance3 = 8 # second path second leg
      zup = .375
      # inches
      wd1 = welddistance1 * 25.4 / 1000
      wd2 = welddistance2 * 25.4 / 1000
      wd3 = welddistance3 * 25.4 / 1000
      zup = zup * 25.4 / 1000
      chamferovermm =  chamferover * 25.4 / 1000

      x = pointintersect[0] + l1delxunit * chamferovermm
      y = pointintersect[1] + l1delyunit * chamferovermm
      z = pointintersect[2] + zup

      #apply actual rxryrz to points
      # convert the headings to rxryrz and insert those values into the relevant points
      rxryrz = convert_heading_to_axang_preheatdown(heading1)
      rx = rxryrz[0]
      ry = rxryrz[1]
      rz = rxryrz[2]

      point1 = p[x + wd1*listleans[0], y + wd1*listleans[1], z + wd1, rx, ry, rz] # add in the listleans factor to follow the face of the box as we move up
      point2 = p[x, y, z, rx, ry, rz]

      # convert the headings to rxryrz and insert those values into the relevant points
      rxryrz = convert_heading_to_axang_ccw(heading1)
      rx = rxryrz[0]
      ry = rxryrz[1]
      rz = rxryrz[2]

      point4 = p[x, y, z, rx, ry, rz]
      x = x + l1delxunit * wd2
      y = y + l1delyunit * wd2
      point5 = p[x, y, z, rx, ry, rz]

      # FIND THE POINTS ON THE LINES OF THE SECOND AROUND PATH
      roundoverdistance = 0.05
      rod = roundoverdistance * 25.4 / 1000

      # now we have the unit vector. extend the weld distance from the intersection
      x = pointintersect[0] + l1delxunit * chamferovermm
      y = pointintersect[1] + l1delyunit * chamferovermm
      # convert the headings to rxryrz and insert those values into the relevant points
      rxryrz = convert_heading_to_axang(heading1)
      rx = rxryrz[0]
      ry = rxryrz[1]
      rz = rxryrz[2]
      point_1 = p[x, y, z, rx, ry, rz]

      x = pointintersect[0] + l1delxunit * rod
      y = pointintersect[1] + l1delyunit * rod
      point_2 = p[x, y, z, rx, ry, rz]

      # now we have the unit vector. extend the weld distance from the intersection
      x = pointintersect[0] + l2delxunit * wd3
      y = pointintersect[1] + l2delyunit * wd3
      # convert the headings to rxryrz and insert those values into the relevant points
      rxryrz = convert_heading_to_axang(heading3)
      rx = rxryrz[0]
      ry = rxryrz[1]
      rz = rxryrz[2]
      point_5 = p[x, y, z, rx, ry, rz]

      x = pointintersect[0] + l2delxunit * rod
      y = pointintersect[1] + l2delyunit * rod
      point_4 = p[x, y, z, rx, ry, rz]

      #FIND POINT 3
      # by calling analyze_touchpoints()
      atret = analyze_touchpoints(point_2, point_1, point_4, point_5, pointintersect)
      point_3 = atret[5]


      struct2 = struct(point1=point1, point2=point2, point4=point4, point5=point5, point_1=point_1, point_2=point_2, point_3=point_3, point_4=point_4, point_5=point_5)
      return struct2
  end

  # given a struct from analyze_touchpoints_only(), calculate the points
  # for left, for non-extended
  def calculate_DOtA_points_left(struct1, listleans, chamferover):
      # get the stuff from the struct
      pointintersect = struct1[0]
      heading1 = struct1[1]
      heading2 = struct1[2]
      heading3 = struct1[3]
      l1delxunit = struct1[4]
      l1delyunit = struct1[5]
      l2delxunit = struct1[6]
      l2delyunit = struct1[7]

      # FIND THE POINTS ON THE LINES OF THE FIRST TURN PATH
      # find locations 8 inches away from  intersect point
      # CONST
      welddistance1 = 8 # vertical weld distance
      welddistance2 = 6 # first path second leg
      welddistance3 = 8 # second path second leg
      zup = .375
      # inches
      wd1 = welddistance1 * 25.4 / 1000
      wd2 = welddistance2 * 25.4 / 1000
      wd3 = welddistance3 * 25.4 / 1000
      zup = zup * 25.4 / 1000
      chamferovermm =  chamferover * 25.4 / 1000

      x = pointintersect[0] + l2delxunit * chamferovermm
      y = pointintersect[1] + l2delyunit * chamferovermm
      z = pointintersect[2] + zup

      #apply actual rxryrz to points
      # convert the headings to rxryrz and insert those values into the relevant points
      rxryrz = convert_heading_to_axang_preheatdown(heading3)
      rx = rxryrz[0]
      ry = rxryrz[1]
      rz = rxryrz[2]

      point1 = p[x + wd1*listleans[0], y + wd1*listleans[1], z + wd1, rx, ry, rz]
      point2 = p[x, y, z, rx, ry, rz]

      # convert the headings to rxryrz and insert those values into the relevant points
      rxryrz = convert_heading_to_axang(heading3)
      rx = rxryrz[0]
      ry = rxryrz[1]
      rz = rxryrz[2]

      point4 = p[x, y, z, rx, ry, rz]
      x = x + l2delxunit * wd2
      y = y + l2delyunit * wd2
      point5 = p[x, y, z, rx, ry, rz]

      # FIND THE POINTS ON THE LINES OF THE SECOND AROUND PATH
      roundoverdistance = 0.05
      rod = roundoverdistance * 25.4 / 1000

      # now we have the unit vector. extend the weld distance from the intersection
      x = pointintersect[0] + l2delxunit * chamferovermm
      y = pointintersect[1] + l2delyunit * chamferovermm
      # convert the headings to rxryrz and insert those values into the relevant points
      rxryrz = convert_heading_to_axang_ccw(heading3)
      rx = rxryrz[0]
      ry = rxryrz[1]
      rz = rxryrz[2]
      point_1 = p[x, y, z, rx, ry, rz]

      x = pointintersect[0] + l2delxunit * rod
      y = pointintersect[1] + l2delyunit * rod
      point_2 = p[x, y, z, rx, ry, rz]

      # now we have the unit vector. extend the weld distance from the intersection
      x = pointintersect[0] + l1delxunit * wd3
      y = pointintersect[1] + l1delyunit * wd3
      # convert the headings to rxryrz and insert those values into the relevant points
      rxryrz = convert_heading_to_axang_ccw(heading1)
      rx = rxryrz[0]
      ry = rxryrz[1]
      rz = rxryrz[2]
      point_5 = p[x, y, z, rx, ry, rz]

      x = pointintersect[0] + l1delxunit * rod
      y = pointintersect[1] + l1delyunit * rod
      point_4 = p[x, y, z, rx, ry, rz]

      #FIND POINT 3
      # by calling analyze_touchpoints()
      atret = analyze_touchpoints(point_2, point_1, point_4, point_5, pointintersect)
      point_3 = atret[5]
      #point 3 will not have the correct rxryrz though because now the gun needs to be face up.
      rxryrz = convert_heading_to_axang_ccw(heading2)
      rx = rxryrz[0]
      ry = rxryrz[1]
      rz = rxryrz[2]
      point_3 = p[point_3[0], point_3[1], point_3[2], rx, ry, rz]

      struct2 = struct(point1=point1, point2=point2, point4=point4, point5=point5, point_1=point_1, point_2=point_2, point_3=point_3, point_4=point_4, point_5=point_5)
      return struct2
  end

  # given a struct from analyze_touchpoints_only(), calculate the points
  # for right, for extended
  def calculate_DOtA_points_right_extended(struct1, listleans, chamferover, chamferup, tcp_pose_top):
      # get the stuff from the struct
      pointintersect = struct1[0]
      heading1 = struct1[1]
      heading2 = struct1[2]
      heading3 = struct1[3]
      l1delxunit = struct1[4]
      l1delyunit = struct1[5]
      l2delxunit = struct1[6]
      l2delyunit = struct1[7]

      # FIND THE POINTS ON THE LINES OF THE FIRST TURN PATH
      # find locations 8 inches away from  intersect point
      # CONST
      # welddistance1 = 8 # vertical weld distance
      welddistance2 = 6 # first path second leg
      welddistance3 = 8 # second path second leg

      # inches
      # wd1 = welddistance1 * 25.4 / 1000
      wd2 = welddistance2 * 25.4 / 1000
      wd3 = welddistance3 * 25.4 / 1000
      zup = chamferup * 25.4 / 1000
      chamferovermm =  chamferover * 25.4 / 1000

      # weld distance is the distance that it will weld. this will make it start at the z height that the user specified
      wd1 = tcp_pose_top[2] - pointintersect[2] - zup

      x = pointintersect[0] + l1delxunit * chamferovermm
      y = pointintersect[1] + l1delyunit * chamferovermm
      z = pointintersect[2] + zup

      #apply actual rxryrz to points
      # convert the headings to rxryrz and insert those values into the relevant points
      rxryrz = convert_heading_to_axang_preheatdown(heading1)
      rx = rxryrz[0]
      ry = rxryrz[1]
      rz = rxryrz[2]

      point1 = p[x + wd1*listleans[0], y + wd1*listleans[1], z + wd1, rx, ry, rz] # add in the listleans factor to follow the face of the box as we move up
      point2 = p[x, y, z, rx, ry, rz]

      # convert the headings to rxryrz and insert those values into the relevant points
      rxryrz = convert_heading_to_axang_ccw(heading1)
      rx = rxryrz[0]
      ry = rxryrz[1]
      rz = rxryrz[2]

      point4 = p[x, y, z, rx, ry, rz]
      x = x + l1delxunit * wd2
      y = y + l1delyunit * wd2
      point5 = p[x, y, z, rx, ry, rz]

      # FIND THE POINTS ON THE LINES OF THE SECOND AROUND PATH
      roundoverdistance = 0.05
      rod = roundoverdistance * 25.4 / 1000

      # now we have the unit vector. extend the weld distance from the intersection
      x = pointintersect[0] + l1delxunit * chamferovermm
      y = pointintersect[1] + l1delyunit * chamferovermm
      # convert the headings to rxryrz and insert those values into the relevant points
      rxryrz = convert_heading_to_axang(heading1)
      rx = rxryrz[0]
      ry = rxryrz[1]
      rz = rxryrz[2]
      point_1 = p[x, y, z, rx, ry, rz]

      x = pointintersect[0] + l1delxunit * rod
      y = pointintersect[1] + l1delyunit * rod
      point_2 = p[x, y, z, rx, ry, rz]

      # convert the headings to rxryrz and insert those values into the relevant points
      rxryrz = convert_heading_to_axang(heading3)
      rx = rxryrz[0]
      ry = rxryrz[1]
      rz = rxryrz[2]

      x = pointintersect[0] + l2delxunit * rod
      y = pointintersect[1] + l2delyunit * rod
      point_4 = p[x, y, z, rx, ry, rz]

      # now we have the unit vector. extend the weld distance from the intersection
      x = pointintersect[0] + l2delxunit * wd3
      y = pointintersect[1] + l2delyunit * wd3
      point_5 = p[x, y, z, rx, ry, rz]

      #FIND POINT 3
      # by calling analyze_touchpoints()
      atret = analyze_touchpoints(point_2, point_1, point_4, point_5, pointintersect)
      atret5 = atret[5]
      point_3 = p[atret5[0], atret5[1], z, atret5[3], atret5[4], atret5[5]]


      struct2 = struct(point1=point1, point2=point2, point4=point4, point5=point5, point_1=point_1, point_2=point_2, point_3=point_3, point_4=point_4, point_5=point_5)
      return struct2
  end

  # given a struct from analyze_touchpoints_only(), calculate the points
  # for left, for extended
  def calculate_DOtA_points_left_extended(struct1, listleans, chamferover, chamferup, tcp_pose_top):
      # get the stuff from the struct
      pointintersect = struct1[0]
      heading1 = struct1[1]
      heading2 = struct1[2]
      heading3 = struct1[3]
      l1delxunit = struct1[4]
      l1delyunit = struct1[5]
      l2delxunit = struct1[6]
      l2delyunit = struct1[7]

      # FIND THE POINTS ON THE LINES OF THE FIRST TURN PATH
      # find locations 8 inches away from  intersect point
      # CONST
      # welddistance1 = 8 # vertical weld distance
      welddistance2 = 6 # first path second leg
      welddistance3 = 8 # second path second leg

      # inches
      # wd1 = welddistance1 * 25.4 / 1000
      wd2 = welddistance2 * 25.4 / 1000
      wd3 = welddistance3 * 25.4 / 1000
      zup = chamferup * 25.4 / 1000
      chamferovermm =  chamferover * 25.4 / 1000

